C01824=1128.341,-89.185,-46.248,178.702,6.175,149.497
C01825=1128.347,-89.434,-46.238,178.699,6.174,149.498
C01826=1128.352,-89.684,-46.229,178.697,6.174,149.498
C01827=1128.357,-89.934,-46.220,178.696,6.174,149.499
C01828=1128.363,-90.184,-46.210,178.693,6.173,149.499
C01829=1128.368,-90.434,-46.201,178.691,6.172,149.500
C01830=1128.373,-90.683,-46.192,178.690,6.172,149.500
C01831=1128.379,-90.933,-46.182,178.687,6.172,149.501
C01832=1128.384,-91.183,-46.173,178.685,6.171,149.501
C01833=1128.389,-91.433,-46.164,178.683,6.170,149.502
C01834=1128.395,-91.682,-46.154,178.681,6.170,149.502
C01835=1128.400,-91.932,-46.145,178.679,6.169,149.503
C01836=1128.405,-92.182,-46.136,178.677,6.169,149.503
C01837=1128.411,-92.432,-46.127,178.676,6.169,149.504
C01838=1128.416,-92.681,-46.117,178.673,6.168,149.504
C01839=1128.421,-92.930,-46.108,178.671,6.167,149.505
C01840=1128.427,-93.181,-46.099,178.670,6.167,149.505
C01841=1128.433,-93.430,-46.090,178.667,6.166,149.506
C01842=1128.438,-93.680,-46.081,178.665,6.166,149.506
C01843=1128.443,-93.930,-46.071,178.663,6.166,149.507
C01844=1128.448,-94.180,-46.062,178.661,6.165,149.507
C01845=1128.454,-94.430,-46.053,178.659,6.165,149.508
C01846=1128.460,-94.680,-46.044,178.656,6.164,149.508
C01847=1128.465,-94.930,-46.035,178.655,6.164,149.509
C01848=1128.470,-95.179,-46.025,178.653,6.163,149.509
C01849=1128.475,-95.429,-46.016,178.650,6.162,149.510
C01850=1128.481,-95.679,-46.007,178.649,6.162,149.510
C01851=1128.486,-95.929,-45.998,178.647,6.162,149.511
C01852=1128.491,-96.179,-45.989,178.644,6.161,149.511
C01853=1128.497,-96.428,-45.980,178.643,6.161,149.512
C01854=1128.502,-96.677,-45.970,178.641,6.160,149.512
C01855=1128.507,-96.927,-45.961,178.638,6.159,149.513
C01856=1128.513,-97.177,-45.952,178.637,6.160,149.513
C01857=1128.518,-97.427,-45.944,178.635,6.159,149.514
C01858=1128.524,-97.677,-45.934,178.632,6.158,149.514
C01859=1128.529,-97.927,-45.925,178.631,6.158,149.514
C01860=1128.534,-98.177,-45.916,178.629,6.157,149.515
C01861=1128.539,-98.427,-45.907,178.627,6.157,149.515
C01862=1128.546,-98.676,-45.898,178.625,6.157,149.516
C01863=1128.551,-98.926,-45.889,178.623,6.156,149.516
C01864=1128.556,-99.175,-45.880,178.621,6.155,149.517
C01865=1128.561,-99.425,-45.871,178.619,6.155,149.517
C01866=1128.566,-99.675,-45.862,178.617,6.154,149.518
C01867=1128.572,-99.925,-45.852,178.615,6.154,149.518
C01868=1128.577,-100.175,-45.844,178.613,6.154,149.519
C01869=1128.583,-100.424,-45.835,178.611,6.153,149.519
C01870=1128.588,-100.674,-45.826,178.609,6.152,149.520
C01871=1128.593,-100.924,-45.817,178.607,6.152,149.520
C01872=1128.598,-101.173,-45.808,178.605,6.152,149.521
C01873=1128.604,-101.424,-45.799,178.603,6.151,149.521
C01874=1128.609,-101.673,-45.790,178.601,6.151,149.522
C01875=1128.615,-101.923,-45.781,178.599,6.150,149.522
C01876=1128.620,-102.172,-45.772,178.597,6.150,149.523
C01877=1128.626,-102.422,-45.764,178.595,6.149,149.523
C01878=1128.631,-102.672,-45.755,178.593,6.149,149.524
C01879=1128.637,-102.945,-45.745,178.591,6.148,149.524
C01880=1128.642,-103.217,-45.736,178.589,6.148,149.525
C01881=1128.648,-103.489,-45.725,178.586,6.148,149.525
C01882=1128.654,-103.762,-45.715,178.584,6.147,149.526
C01883=1128.660,-104.011,-45.707,178.582,6.146,149.526
C01884=1128.665,-104.261,-45.698,178.580,6.146,149.527
C01885=1128.670,-104.511,-45.689,178.578,6.145,149.527
C01886=1128.676,-104.761,-45.680,178.577,6.145,149.528
C01887=1128.681,-105.011,-45.671,178.574,6.145,149.528
C01888=1128.687,-105.260,-45.663,178.572,6.144,149.529
C01889=1128.692,-105.510,-45.654,178.571,6.144,149.529
C01890=1128.697,-105.760,-45.646,178.568,6.143,149.530
C01891=1128.702,-106.010,-45.637,178.566,6.143,149.530
C01892=1128.708,-106.260,-45.628,178.565,6.143,149.531
C01893=1128.713,-106.509,-45.619,178.562,6.142,149.531
C01894=1128.718,-106.759,-45.610,178.561,6.142,149.532
C01895=1128.724,-107.009,-45.601,178.559,6.141,149.532
C01896=1128.730,-107.259,-45.592,178.556,6.140,149.533
C01897=1128.736,-107.509,-45.584,178.555,6.140,149.533
C01898=1128.741,-107.758,-45.575,178.553,6.140,149.534
C01899=1128.746,-108.008,-45.566,178.551,6.140,149.534
C01900=1128.751,-108.258,-45.557,178.549,6.139,149.535
C01901=1128.757,-108.507,-45.549,178.547,6.138,149.535
C01902=1128.762,-108.757,-45.540,178.545,6.138,149.535
C01903=1128.768,-109.008,-45.532,178.543,6.137,149.536
C01904=1128.773,-109.257,-45.523,178.541,6.136,149.536
C01905=1128.778,-109.507,-45.514,178.539,6.136,149.537
C01906=1128.784,-109.756,-45.506,178.537,6.136,149.537
C01907=1128.789,-110.006,-45.497,178.536,6.136,149.538
C01908=1128.794,-110.257,-45.488,178.533,6.135,149.538
C01909=1128.800,-110.506,-45.480,178.531,6.134,149.539
C01910=1128.805,-110.756,-45.471,178.530,6.134,149.539
C01911=1128.810,-111.006,-45.462,178.527,6.134,149.540
C01912=1128.816,-111.255,-45.454,178.526,6.134,149.540
C01913=1128.822,-111.505,-45.445,178.524,6.133,149.541
C01914=1128.827,-111.755,-45.436,178.521,6.132,149.541
C01915=1128.832,-112.005,-45.428,178.520,6.132,149.542
C01916=1128.838,-112.255,-45.420,178.518,6.131,149.542
C01917=1128.842,-112.504,-45.411,178.516,6.132,149.543
C01918=1128.848,-112.754,-45.403,178.514,6.131,149.543
C01919=1128.853,-113.003,-45.394,178.512,6.131,149.544
C01920=1128.859,-113.254,-45.386,178.510,6.130,149.544
C01921=1128.864,-113.504,-45.377,178.508,6.129,149.545
C01922=1128.870,-113.753,-45.368,178.506,6.129,149.545
C01923=1128.875,-114.003,-45.360,178.505,6.128,149.545
C01924=1128.880,-114.253,-45.351,178.503,6.128,149.546
C01925=1128.886,-114.502,-45.343,178.501,6.128,149.546
C01926=1128.892,-114.753,-45.335,178.499,6.127,149.547
C01927=1128.897,-115.003,-45.326,178.497,6.127,149.547
C01928=1128.903,-115.252,-45.317,178.495,6.126,149.548
C01929=1128.908,-115.502,-45.309,178.493,6.126,149.548
C01930=1128.913,-115.752,-45.300,178.491,6.125,149.549
C01931=1128.918,-116.001,-45.292,178.489,6.125,149.549
C01932=1128.924,-116.251,-45.284,178.487,6.125,149.550
C01933=1128.929,-116.501,-45.275,178.485,6.124,149.550
C01934=1128.935,-116.750,-45.267,178.483,6.124,149.551
C01935=1128.940,-117.001,-45.258,178.481,6.123,149.551
C01936=1128.945,-117.251,-45.249,178.480,6.123,149.552
C01937=1128.951,-117.500,-45.242,178.478,6.122,149.552
C01938=1128.957,-117.750,-45.233,178.476,6.122,149.552
C01939=1128.961,-118.000,-45.224,178.474,6.122,149.553
C01940=1128.967,-118.250,-45.217,178.472,6.121,149.553
C01941=1128.972,-118.499,-45.208,178.470,6.121,149.554
C01942=1128.978,-118.749,-45.200,178.468,6.120,149.554
C01943=1128.983,-118.999,-45.191,178.467,6.120,149.555
C01944=1128.989,-119.250,-45.183,178.464,6.119,149.555
C01945=1128.994,-119.498,-45.175,178.463,6.119,149.556
C01946=1128.999,-119.748,-45.166,178.461,6.119,149.556
C01947=1129.005,-119.999,-45.158,178.459,6.119,149.557
C01948=1129.010,-120.248,-45.149,178.457,6.118,149.557
C01949=1129.016,-120.498,-45.141,178.455,6.117,149.558
C01950=1129.021,-120.747,-45.133,178.453,6.117,149.558
C01951=1129.026,-120.998,-45.125,178.451,6.116,149.559
C01952=1129.032,-121.247,-45.116,178.450,6.116,149.559
C01953=1129.038,-121.497,-45.108,178.447,6.116,149.560
C01954=1129.043,-121.747,-45.099,178.446,6.116,149.560
C01955=1129.048,-121.997,-45.092,178.444,6.115,149.561
C01956=1129.053,-122.246,-45.083,178.442,6.115,149.561
C01957=1129.059,-122.496,-45.075,178.440,6.114,149.562
C01958=1129.064,-122.746,-45.067,178.439,6.114,149.562
C01959=1129.069,-122.996,-45.059,178.436,6.113,149.562
C01960=1129.075,-123.245,-45.050,178.434,6.112,149.563
C01961=1129.080,-123.496,-45.042,178.433,6.112,149.563
C01962=1129.086,-123.745,-45.034,178.430,6.112,149.564
C01963=1129.091,-123.995,-45.026,178.429,6.112,149.564
C01964=1129.097,-124.245,-45.018,178.427,6.111,149.565
C01965=1129.102,-124.495,-45.009,178.425,6.111,149.565
C01966=1129.108,-124.745,-45.001,178.423,6.110,149.565
C01967=1129.113,-124.994,-44.993,178.422,6.110,149.566
C01968=1129.118,-125.244,-44.985,178.420,6.109,149.566
C01969=1129.124,-125.494,-44.977,178.418,6.109,149.567
C01970=1129.129,-125.744,-44.969,178.416,6.109,149.567
C01971=1129.135,-125.994,-44.961,178.414,6.109,149.568
C01972=1129.140,-126.243,-44.952,178.412,6.108,149.568
C01973=1129.146,-126.493,-44.944,178.410,6.108,149.569
C01974=1129.151,-126.743,-44.937,178.409,6.107,149.569
C01975=1129.156,-126.992,-44.928,178.407,6.107,149.570
C01976=1129.162,-127.243,-44.920,178.405,6.106,149.570
C01977=1129.167,-127.492,-44.912,178.403,6.106,149.571
C01978=1129.172,-127.742,-44.904,178.401,6.105,149.571
C01979=1129.179,-127.992,-44.896,178.400,6.105,149.572
C01980=1129.183,-128.242,-44.888,178.397,6.105,149.572
C01981=1129.189,-128.491,-44.880,178.396,6.104,149.572
C01982=1129.195,-128.742,-44.872,178.394,6.104,149.573
C01983=1128.773,-128.753,-44.916,178.391,6.108,149.575
C01984=1128.768,-128.503,-44.925,178.392,6.108,149.574
C01985=1128.762,-128.253,-44.933,178.395,6.108,149.574
C01986=1128.757,-128.003,-44.940,178.396,6.108,149.573
C01987=1128.752,-127.754,-44.949,178.398,6.109,149.573
C01988=1128.746,-127.504,-44.957,178.399,6.109,149.572
C01989=1128.741,-127.254,-44.964,178.402,6.110,149.572
C01990=1128.736,-127.004,-44.973,178.403,6.110,149.571
C01991=1128.730,-126.754,-44.981,178.405,6.111,149.571
C01992=1128.725,-126.504,-44.989,178.407,6.111,149.570
C01993=1128.719,-126.255,-44.997,178.409,6.111,149.570
C01994=1128.714,-126.005,-45.005,178.411,6.111,149.570
C01995=1128.708,-125.755,-45.013,178.413,6.113,149.569
C01996=1128.703,-125.505,-45.021,178.414,6.113,149.569
C01997=1128.697,-125.256,-45.029,178.416,6.113,149.568
C01998=1128.692,-125.006,-45.038,178.418,6.113,149.568
C01999=1128.687,-124.756,-45.046,178.420,6.114,149.567
C02000=1128.681,-124.506,-45.054,178.422,6.114,149.567
C02001=1128.676,-124.256,-45.062,178.424,6.115,149.566
C02002=1128.670,-124.006,-45.070,178.425,6.115,149.566
C02003=1128.665,-123.757,-45.079,178.427,6.116,149.566
C02004=1128.659,-123.507,-45.086,178.429,6.116,149.565
C02005=1128.654,-123.257,-45.095,178.431,6.116,149.565
C02006=1128.648,-123.007,-45.103,178.433,6.117,149.564
C02007=1128.644,-122.758,-45.111,178.435,6.117,149.564
C02008=1128.638,-122.507,-45.120,178.437,6.118,149.563
C02009=1128.632,-122.258,-45.128,178.439,6.118,149.563
C02010=1128.627,-122.008,-45.136,178.441,6.119,149.562
C02011=1128.622,-121.759,-45.144,178.442,6.119,149.562
C02012=1128.617,-121.508,-45.152,178.444,6.120,149.561
C02013=1128.611,-121.258,-45.161,178.446,6.120,149.561
C02014=1128.605,-121.009,-45.169,178.448,6.120,149.560
C02015=1128.601,-120.759,-45.177,178.450,6.121,149.560
C02016=1128.595,-120.509,-45.185,178.452,6.121,149.559
C02017=1128.590,-120.260,-45.194,178.454,6.122,149.559
C02018=1128.584,-120.009,-45.202,178.456,6.122,149.558
C02019=1128.578,-119.760,-45.211,178.458,6.122,149.558
C02020=1128.573,-119.509,-45.219,178.459,6.123,149.558
C02021=1128.568,-119.261,-45.227,178.461,6.124,149.557
C02022=1128.562,-119.010,-45.235,178.463,6.123,149.557
C02023=1128.557,-118.760,-45.244,178.465,6.124,149.556
C02024=1128.551,-118.511,-45.253,178.467,6.125,149.556
C02025=1128.546,-118.261,-45.261,178.469,6.125,149.555
C02026=1128.542,-118.011,-45.269,178.471,6.126,149.555
C02027=1128.535,-117.761,-45.277,178.472,6.126,149.554
C02028=1128.530,-117.512,-45.286,178.475,6.126,149.554
C02029=1128.524,-117.262,-45.294,178.476,6.126,149.553
C02030=1128.519,-117.012,-45.303,178.478,6.127,149.553
C02031=1128.514,-116.762,-45.311,178.480,6.127,149.553
C02032=1128.508,-116.512,-45.319,178.482,6.128,149.552
C02033=1128.503,-116.262,-45.328,178.484,6.129,149.552
C02034=1128.498,-116.013,-45.336,178.486,6.129,149.551
C02035=1128.492,-115.763,-45.344,178.488,6.130,149.551
C02036=1128.487,-115.513,-45.353,178.489,6.129,149.550
C02037=1128.482,-115.263,-45.361,178.492,6.130,149.550
C02038=1128.476,-115.014,-45.370,178.493,6.130,149.549
C02039=1128.471,-114.764,-45.379,178.495,6.131,149.549
C02040=1128.465,-114.513,-45.387,178.498,6.132,149.548
C02041=1128.459,-114.264,-45.395,178.499,6.132,149.548
C02042=1128.454,-114.014,-45.404,178.501,6.132,149.547
C02043=1128.449,-113.764,-45.413,178.503,6.132,149.547
C02044=1128.443,-113.515,-45.421,178.505,6.133,149.546
C02045=1128.438,-113.265,-45.430,178.507,6.134,149.546
C02046=1128.433,-113.015,-45.438,178.508,6.134,149.546
C02047=1128.427,-112.766,-45.446,178.511,6.135,149.545
C02048=1128.422,-112.516,-45.455,178.512,6.135,149.545
C02049=1128.417,-112.266,-45.464,178.514,6.136,149.544
C02050=1128.411,-112.016,-45.472,178.516,6.136,149.544
C02051=1128.406,-111.766,-45.481,178.518,6.136,149.543
C02052=1128.401,-111.516,-45.490,178.520,6.137,149.543
C02053=1128.395,-111.267,-45.498,178.522,6.137,149.542
C02054=1128.389,-111.017,-45.506,178.524,6.138,149.542
C02055=1128.384,-110.767,-45.515,178.526,6.138,149.541
C02056=1128.379,-110.517,-45.524,178.528,6.138,149.541
C02057=1128.373,-110.268,-45.533,178.530,6.139,149.540
C02058=1128.368,-110.018,-45.541,178.532,6.139,149.540
C02059=1128.363,-109.768,-45.550,178.534,6.140,149.539
C02060=1128.357,-109.518,-45.559,178.536,6.140,149.539
C02061=1128.352,-109.269,-45.567,178.538,6.141,149.538
C02062=1128.346,-109.019,-45.576,178.540,6.141,149.538
C02063=1128.341,-108.769,-45.585,178.542,6.141,149.537
C02064=1128.336,-108.518,-45.593,178.544,6.142,149.537
C02065=1128.330,-108.269,-45.602,178.546,6.143,149.536
C02066=1128.325,-108.019,-45.610,178.547,6.143,149.536
C02067=1128.320,-107.770,-45.619,178.549,6.144,149.536
C02068=1128.315,-107.520,-45.628,178.551,6.144,149.535
C02069=1128.309,-107.271,-45.637,178.553,6.144,149.535
C02070=1128.303,-107.020,-45.645,178.555,6.145,149.534
C02071=1128.298,-106.770,-45.654,178.557,6.145,149.534
C02072=1128.293,-106.520,-45.663,178.559,6.146,149.533
C02073=1128.287,-106.271,-45.671,178.561,6.146,149.533
C02074=1128.282,-106.021,-45.680,178.563,6.147,149.532
C02075=1128.276,-105.771,-45.690,178.565,6.147,149.532
C02076=1128.271,-105.521,-45.699,178.567,6.147,149.531
C02077=1128.266,-105.272,-45.707,178.569,6.148,149.531
C02078=1128.260,-105.022,-45.716,178.571,6.149,149.530
C02079=1128.255,-104.772,-45.724,178.573,6.149,149.530
C02080=1128.249,-104.522,-45.733,178.575,6.149,149.529
C02081=1128.244,-104.272,-45.742,178.576,6.149,149.529
C02082=1128.239,-104.022,-45.751,178.579,6.150,149.528
C02083=1128.233,-103.773,-45.759,178.581,6.151,149.528
C02084=1128.228,-103.501,-45.769,178.583,6.152,149.527
C02085=1128.222,-103.229,-45.779,178.585,6.152,149.527
C02086=1128.216,-102.956,-45.789,178.587,6.152,149.526
C02087=1128.210,-102.684,-45.798,178.590,6.153,149.526
C02088=1128.205,-102.433,-45.808,178.592,6.153,149.525
C02089=1128.199,-102.184,-45.817,178.593,6.153,149.525
C02090=1128.194,-101.934,-45.825,178.596,6.154,149.524
C02091=1128.188,-101.685,-45.834,178.597,6.154,149.524
C02092=1128.183,-101.435,-45.843,178.599,6.155,149.523
C02093=1128.178,-101.185,-45.852,178.602,6.156,149.523
C02094=1128.173,-100.935,-45.861,178.603,6.156,149.522
C02095=1128.167,-100.685,-45.870,178.605,6.156,149.522
C02096=1128.162,-100.435,-45.879,178.608,6.157,149.521
C02097=1128.156,-100.186,-45.888,178.609,6.157,149.521
C02098=1128.151,-99.936,-45.897,178.611,6.158,149.520
C02099=1128.146,-99.686,-45.905,178.614,6.158,149.520
C02100=1128.140,-99.436,-45.915,178.615,6.158,149.519
C02101=1128.135,-99.186,-45.924,178.617,6.159,149.519
C02102=1128.130,-98.937,-45.933,178.620,6.160,149.518
C02103=1128.125,-98.687,-45.942,178.621,6.160,149.518
C02104=1128.119,-98.438,-45.951,178.623,6.161,149.517
C02105=1128.113,-98.188,-45.960,178.626,6.161,149.517
C02106=1128.108,-97.938,-45.969,178.627,6.161,149.516
C02107=1128.103,-97.688,-45.978,178.629,6.162,149.516
C02108=1128.097,-97.438,-45.987,178.631,6.163,149.515
C02109=1128.092,-97.188,-45.996,178.633,6.163,149.515
C02110=1128.086,-96.938,-46.005,178.635,6.164,149.514
C02111=1128.081,-96.688,-46.014,178.637,6.164,149.514
C02112=1128.076,-96.440,-46.024,178.639,6.164,149.513
C02113=1128.071,-96.190,-46.032,178.641,6.165,149.513
C02114=1128.065,-95.940,-46.042,178.643,6.166,149.512
C02115=1128.060,-95.690,-46.051,178.645,6.166,149.512
C02116=1128.054,-95.440,-46.060,178.647,6.166,149.511
C02117=1128.048,-95.190,-46.069,178.649,6.167,149.511
C02118=1128.043,-94.940,-46.078,178.651,6.167,149.510
C02119=1128.038,-94.691,-46.088,178.653,6.168,149.510
C02120=1128.033,-94.441,-46.097,178.655,6.169,149.509
C02121=1128.027,-94.191,-46.106,178.657,6.169,149.509
C02122=1128.022,-93.941,-46.115,178.659,6.169,149.509
C02123=1128.017,-93.691,-46.124,178.661,6.170,149.508
C02124=1128.011,-93.442,-46.134,178.664,6.171,149.508
C02125=1128.006,-93.192,-46.143,178.665,6.171,149.507
C02126=1128.001,-92.943,-46.152,178.667,6.172,149.507
C02127=1127.995,-92.692,-46.161,178.670,6.172,149.506
C02128=1127.990,-92.443,-46.171,178.672,6.172,149.505
C02129=1127.985,-92.193,-46.180,178.674,6.173,149.505
C02130=1127.979,-91.943,-46.189,178.676,6.173,149.504
C02131=1127.974,-91.693,-46.198,178.678,6.173,149.504
C02132=1127.969,-91.444,-46.208,178.680,6.174,149.503
C02133=1127.963,-91.194,-46.217,178.682,6.175,149.503
C02134=1127.958,-90.944,-46.226,178.684,6.176,149.502
C02135=1127.952,-90.694,-46.235,178.686,6.176,149.502
C02136=1127.947,-90.445,-46.245,178.688,6.176,149.502
C02137=1127.942,-90.195,-46.254,178.690,6.177,149.501
C02138=1127.936,-89.945,-46.263,178.692,6.177,149.501
C02139=1127.931,-89.695,-46.273,178.694,6.178,149.500
C02140=1127.926,-89.446,-46.282,178.696,6.178,149.500
C02141=1127.921,-89.196,-46.291,178.698,6.179,149.499
C02142=1127.915,-88.946,-46.301,178.700,6.179,149.499
C02143=1127.910,-88.696,-46.310,178.702,6.180,149.498
C02144=1127.904,-88.446,-46.320,178.704,6.181,149.498
C02145=1127.899,-88.197,-46.329,178.706,6.181,149.497
C02146=1127.894,-87.947,-46.338,178.708,6.181,149.497
C02147=1127.888,-87.697,-46.348,178.711,6.182,149.496
C02148=1127.883,-87.448,-46.357,178.713,6.182,149.495
C02149=1127.877,-87.198,-46.367,178.715,6.182,149.495
C02150=1127.872,-86.948,-46.376,178.717,6.183,149.494
C02151=1127.866,-86.698,-46.386,178.719,6.184,149.494
C02152=1127.861,-86.448,-46.395,178.721,6.184,149.494
C02153=1127.856,-86.199,-46.404,178.723,6.185,149.493
C02154=1127.850,-85.949,-46.414,178.725,6.185,149.493
C02155=1127.846,-85.700,-46.423,178.727,6.186,149.492
C02156=1127.840,-85.449,-46.433,178.729,6.186,149.492
C02157=1127.835,-85.200,-46.443,178.731,6.187,149.491
C02158=1127.830,-84.949,-46.452,178.733,6.188,149.491
C02159=1127.824,-84.700,-46.461,178.735,6.188,149.490
C02160=1127.819,-84.450,-46.471,178.737,6.188,149.490
C02161=1127.814,-84.200,-46.480,178.740,6.189,149.489
C02162=1127.808,-83.951,-46.491,178.742,6.189,149.488
C02163=1127.803,-83.701,-46.499,178.744,6.190,149.488
C02164=1127.797,-83.451,-46.510,178.746,6.190,149.487
C02165=1127.792,-83.201,-46.519,178.748,6.191,149.487
C02166=1127.786,-82.952,-46.529,178.750,6.192,149.487
C02167=1127.781,-82.702,-46.538,178.752,6.192,149.486
C02168=1127.776,-82.452,-46.548,178.754,6.192,149.486
C02169=1127.771,-82.203,-46.557,178.756,6.193,149.485
C02170=1127.766,-81.952,-46.567,178.758,6.194,149.485
C02171=1127.760,-81.702,-46.576,178.760,6.195,149.484
C02172=1127.755,-81.453,-46.586,178.763,6.194,149.483
C02173=1127.750,-81.203,-46.595,178.765,6.195,149.483
C02174=1127.744,-80.954,-46.606,178.767,6.196,149.482
C02175=1127.739,-80.704,-46.615,178.769,6.196,149.482
C02176=1127.733,-80.454,-46.625,178.771,6.196,149.481
C02177=1127.728,-80.205,-46.635,178.773,6.197,149.481
C02178=1127.723,-79.955,-46.644,178.775,6.198,149.480
C02179=1127.718,-79.705,-46.654,178.777,6.199,149.480
C02180=1127.713,-79.455,-46.664,178.779,6.199,149.480
C02181=1127.707,-79.205,-46.673,178.781,6.199,149.479
C02182=1127.702,-78.956,-46.683,178.783,6.200,149.479
C02183=1127.696,-78.706,-46.693,178.786,6.201,149.478
C02184=1127.690,-78.456,-46.703,178.788,6.201,149.477
C02185=1127.686,-78.207,-46.712,178.790,6.201,149.477
C02186=1127.680,-77.957,-46.722,178.792,6.202,149.476
C02187=1127.675,-77.707,-46.732,178.794,6.203,149.476
C02188=1127.669,-77.435,-46.742,178.796,6.204,149.475
C02189=1127.663,-77.164,-46.753,178.799,6.204,149.475
C02190=1127.657,-76.892,-46.764,178.801,6.205,149.474
C02191=1127.652,-76.621,-46.775,178.803,6.205,149.474
C02192=1127.646,-76.370,-46.784,178.805,6.205,149.473
C02193=1127.641,-76.121,-46.794,178.807,6.206,149.473
C02194=1127.636,-75.872,-46.804,178.809,6.207,149.472
C02195=1127.630,-75.621,-46.814,178.812,6.207,149.472
C02196=1127.621,-75.201,-46.831,178.815,6.208,149.471
C02197=1127.594,-73.952,-46.879,179.491,4.912,148.990
C02198=1127.589,-73.702,-46.889,179.491,4.918,148.991
C02199=1127.584,-73.452,-46.898,179.492,4.923,148.992
C02200=1127.578,-73.203,-46.908,179.492,4.928,148.993
C02201=1127.573,-72.953,-46.917,179.492,4.934,148.994
C02202=1127.567,-72.703,-46.927,179.493,4.939,148.995
C02203=1127.563,-72.453,-46.937,179.493,4.945,148.996
C02204=1127.557,-72.203,-46.947,179.493,4.950,148.998
C02205=1127.551,-71.953,-46.956,179.493,4.955,148.999
C02206=1127.546,-71.704,-46.966,179.494,4.961,149.000
C02207=1127.540,-71.454,-46.975,179.494,4.965,149.001
C02208=1127.535,-71.205,-46.985,179.494,4.971,149.002
C02209=1127.530,-70.955,-46.995,179.495,4.976,149.003
C02210=1127.525,-70.705,-47.004,179.495,4.981,149.004
C02211=1127.519,-70.456,-47.014,179.495,4.987,149.005
C02212=1127.514,-70.205,-47.024,179.496,4.992,149.006
C02213=1127.509,-69.956,-47.034,179.497,4.998,149.007
C02214=1127.503,-69.706,-47.044,179.496,5.003,149.008
C02215=1127.497,-69.456,-47.053,179.497,5.008,149.009
C02216=1127.493,-69.207,-47.063,179.497,5.014,149.010
C02217=1127.487,-68.957,-47.073,179.498,5.019,149.011
C02218=1127.481,-68.707,-47.083,179.498,5.024,149.012
C02219=1127.477,-68.457,-47.093,179.499,5.030,149.013
C02220=1127.471,-68.207,-47.103,179.499,5.035,149.014
C02221=1127.466,-67.958,-47.113,179.500,5.041,149.015
C02222=1127.460,-67.708,-47.122,179.500,5.045,149.016
C02223=1127.455,-67.458,-47.132,179.501,5.051,149.017
C02224=1127.450,-67.208,-47.143,179.502,5.057,149.018
C02225=1127.445,-66.959,-47.152,179.502,5.062,149.019
C02226=1127.439,-66.709,-47.162,179.503,5.067,149.020
C02227=1127.433,-66.459,-47.172,179.503,5.072,149.021
C02228=1127.428,-66.210,-47.182,179.504,5.078,149.022
C02229=1127.424,-65.960,-47.192,179.505,5.084,149.023
C02230=1127.418,-65.710,-47.203,179.505,5.088,149.024
C02231=1127.412,-65.460,-47.212,179.506,5.094,149.025
C02232=1127.407,-65.211,-47.222,179.507,5.099,149.026
C02233=1127.402,-64.961,-47.232,179.507,5.105,149.027
C02234=1127.397,-64.711,-47.242,179.508,5.110,149.028
C02235=1127.391,-64.462,-47.253,179.509,5.116,149.029
C02236=1127.385,-64.212,-47.263,179.509,5.120,149.030
C02237=1127.381,-63.962,-47.273,179.510,5.126,149.030
C02238=1127.375,-63.712,-47.282,179.511,5.132,149.031
C02239=1127.370,-63.462,-47.293,179.512,5.136,149.032
C02240=1127.365,-63.212,-47.303,179.513,5.142,149.033
C02241=1127.359,-62.963,-47.313,179.514,5.148,149.034
C02242=1127.354,-62.713,-47.324,179.515,5.153,149.035
C02243=1127.349,-62.464,-47.333,179.515,5.158,149.036
C02244=1127.344,-62.214,-47.344,179.516,5.163,149.037
C02245=1127.338,-61.964,-47.354,179.517,5.169,149.038
C02246=1127.329,-61.547,-47.372,179.519,5.178,149.039
C02247=1127.321,-61.128,-47.388,179.520,5.187,149.041
C02248=1127.311,-60.711,-47.405,179.522,5.196,149.042
C02249=1127.303,-60.293,-47.423,179.524,5.204,149.043
C02250=1127.297,-60.043,-47.433,179.524,5.210,149.045
C02251=1127.292,-59.794,-47.444,179.523,5.214,149.046
C02252=1127.287,-59.543,-47.454,179.523,5.219,149.047
C02253=1127.281,-59.294,-47.464,179.523,5.223,149.048
C02254=1127.275,-59.044,-47.475,179.523,5.228,149.049
C02255=1127.271,-58.795,-47.486,179.522,5.232,149.050
C02256=1127.265,-58.545,-47.496,179.522,5.237,149.051
C02257=1127.261,-58.295,-47.506,179.522,5.241,149.052
C02258=1127.255,-58.046,-47.516,179.522,5.246,149.053
C02259=1127.250,-57.796,-47.527,179.521,5.251,149.054
C02260=1127.245,-57.546,-47.537,179.522,5.255,149.055
C02261=1127.239,-57.296,-47.547,179.521,5.261,149.056
C02262=1127.234,-57.047,-47.559,179.521,5.265,149.057
C02263=1127.229,-56.797,-47.569,179.521,5.270,149.058
C02264=1127.224,-56.547,-47.579,179.520,5.274,149.059
C02265=1127.218,-56.297,-47.590,179.520,5.279,149.061
C02266=1127.213,-56.048,-47.600,179.520,5.283,149.062
C02267=1127.208,-55.797,-47.610,179.520,5.288,149.063
C02268=1127.202,-55.549,-47.621,179.519,5.293,149.064
C02269=1127.197,-55.298,-47.632,179.520,5.297,149.065
C02270=1127.192,-55.049,-47.642,179.519,5.302,149.066
C02271=1127.187,-54.798,-47.653,179.519,5.307,149.067
C02272=1127.181,-54.550,-47.664,179.519,5.312,149.068
C02273=1127.176,-54.300,-47.674,179.519,5.316,149.069
C02274=1127.170,-54.049,-47.685,179.519,5.321,149.070
C02275=1127.165,-53.800,-47.695,179.518,5.325,149.071
C02276=1127.160,-53.550,-47.706,179.518,5.330,149.072
C02277=1127.154,-53.301,-47.717,179.518,5.335,149.073
C02278=1127.149,-53.051,-47.727,179.518,5.339,149.074
C02279=1127.144,-52.801,-47.737,179.517,5.344,149.076
C02280=1127.139,-52.551,-47.749,179.517,5.349,149.077
C02281=1127.133,-52.302,-47.759,179.517,5.354,149.078
C02282=1127.128,-52.052,-47.770,179.517,5.358,149.079
C02283=1127.123,-51.803,-47.780,179.517,5.363,149.080
C02284=1127.118,-51.552,-47.791,179.516,5.367,149.081
C02285=1127.112,-51.303,-47.801,179.517,5.372,149.082
C02286=1127.107,-51.053,-47.813,179.516,5.377,149.083
C02287=1127.101,-50.803,-47.823,179.516,5.382,149.084
C02288=1127.096,-50.553,-47.834,179.516,5.386,149.085
C02289=1127.091,-50.304,-47.845,179.516,5.391,149.086
C02290=1127.086,-50.054,-47.855,179.516,5.396,149.087
C02291=1127.081,-49.805,-47.866,179.515,5.400,149.089
C02292=1127.076,-49.555,-47.877,179.515,5.405,149.089
C02293=1127.070,-49.305,-47.888,179.515,5.409,149.091
C02294=1127.065,-49.055,-47.899,179.515,5.415,149.092
C02295=1127.059,-48.806,-47.909,179.514,5.418,149.093
C02296=1127.055,-48.556,-47.921,179.514,5.424,149.094
C02297=1127.049,-48.307,-47.931,179.514,5.429,149.095
C02298=1127.044,-48.091,-47.940,179.514,5.433,149.096
C02299=1127.040,-47.875,-47.950,179.514,5.437,149.097
C02300=1127.036,-47.659,-47.959,179.514,5.441,149.098
C02301=1127.031,-47.444,-47.968,179.514,5.445,149.099
C02302=1127.026,-47.228,-47.978,179.513,5.449,149.100
C02303=1127.022,-47.013,-47.987,179.513,5.453,149.100
C02304=1127.017,-46.797,-47.996,179.513,5.456,149.101
C02305=1127.012,-46.582,-48.005,179.513,5.460,149.102
C02306=1127.007,-46.332,-48.017,179.513,5.466,149.103
C02307=1127.002,-46.082,-48.028,179.512,5.470,149.105
C02308=1126.997,-45.833,-48.039,179.512,5.475,149.106
C02309=1126.992,-45.583,-48.049,179.513,5.480,149.107
C02310=1126.986,-45.333,-48.061,179.512,5.484,149.108
C02311=1126.981,-45.083,-48.071,179.512,5.489,149.109
C02312=1126.975,-44.834,-48.082,179.511,5.494,149.110
C02313=1126.970,-44.584,-48.093,179.512,5.498,149.111
C02314=1126.965,-44.334,-48.105,179.511,5.504,149.112
C02315=1126.959,-44.084,-48.115,179.511,5.508,149.113
C02316=1126.955,-43.835,-48.126,179.511,5.513,149.114
C02317=1126.949,-43.585,-48.137,179.511,5.517,149.115
C02318=1126.944,-43.335,-48.148,179.511,5.522,149.116
C02319=1126.939,-43.086,-48.160,179.511,5.527,149.117
C02320=1126.933,-42.836,-48.170,179.513,5.533,149.118
C02321=1126.928,-42.586,-48.182,179.515,5.539,149.119
C02322=1126.922,-42.337,-48.192,179.517,5.545,149.120
C02323=1126.918,-42.087,-48.203,179.518,5.550,149.120
C02324=1126.912,-41.837,-48.215,179.521,5.556,149.121
C02325=1126.907,-41.588,-48.225,179.523,5.562,149.121
C02326=1126.902,-41.338,-48.237,179.524,5.567,149.122
C02327=1126.896,-41.088,-48.249,179.526,5.573,149.123
C02328=1126.891,-40.838,-48.259,179.527,5.579,149.124
C02329=1126.886,-40.589,-48.270,179.529,5.585,149.124
C02330=1126.881,-40.339,-48.282,179.531,5.590,149.125
C02331=1126.875,-40.090,-48.293,179.533,5.595,149.126
C02332=1126.870,-39.839,-48.304,179.534,5.601,149.127
C02333=1126.865,-39.590,-48.315,179.535,5.606,149.127
C02334=1126.860,-39.340,-48.327,179.537,5.611,149.128
C02335=1126.854,-39.091,-48.338,179.538,5.616,149.129
C02336=1126.849,-38.841,-48.350,179.539,5.622,149.129
C02337=1126.844,-38.591,-48.361,179.541,5.627,149.130
C02338=1126.838,-38.342,-48.372,179.542,5.632,149.131
C02339=1126.833,-38.092,-48.383,179.543,5.638,149.132
C02340=1126.828,-37.842,-48.395,179.545,5.643,149.132
C02341=1126.823,-37.592,-48.407,179.546,5.647,149.133
C02342=1126.817,-37.343,-48.418,179.547,5.653,149.134
C02343=1126.812,-37.094,-48.429,179.548,5.657,149.135
C02344=1126.807,-36.844,-48.441,179.549,5.663,149.135
C02345=1126.802,-36.594,-48.453,179.550,5.667,149.136
C02346=1126.796,-36.343,-48.464,179.551,5.672,149.137
C02347=1126.791,-36.094,-48.475,179.552,5.677,149.138
C02348=1126.786,-35.845,-48.487,179.552,5.682,149.139
C02349=1126.781,-35.595,-48.498,179.553,5.686,149.139
C02350=1126.776,-35.345,-48.510,179.554,5.691,149.140
C02351=1126.770,-35.095,-48.522,179.555,5.696,149.141
C02352=1126.765,-34.846,-48.533,179.556,5.701,149.142
C02353=1126.759,-34.596,-48.544,179.556,5.705,149.143
C02354=1126.756,-34.381,-48.555,179.556,5.709,149.143
C02355=1126.751,-34.165,-48.564,179.557,5.712,149.144
C02356=1126.746,-33.950,-48.575,179.558,5.717,149.145
C02357=1126.742,-33.734,-48.585,179.558,5.721,149.146
C02358=1126.738,-33.519,-48.594,179.558,5.724,149.146
C02359=1126.733,-33.304,-48.605,179.558,5.728,149.147
C02360=1126.728,-33.087,-48.615,179.559,5.733,149.148
C02361=1126.723,-32.872,-48.625,179.559,5.736,149.148
C02362=1126.719,-32.623,-48.637,179.559,5.740,149.149
C02363=1126.713,-32.373,-48.648,179.559,5.745,149.150
C02364=1126.709,-32.123,-48.660,179.559,5.749,149.151
C02365=1126.703,-31.873,-48.672,179.560,5.754,149.152
C02366=1126.697,-31.624,-48.683,179.560,5.758,149.153
C02367=1126.693,-31.375,-48.695,179.559,5.761,149.154
C02368=1126.687,-31.125,-48.707,179.559,5.767,149.155
C02369=1126.682,-30.875,-48.719,179.559,5.771,149.156
C02370=1126.676,-30.625,-48.731,179.559,5.774,149.157
C02371=1126.672,-30.375,-48.742,179.559,5.778,149.158
C02372=1126.666,-30.126,-48.754,179.558,5.783,149.159
C02373=1126.661,-29.876,-48.766,179.558,5.787,149.160
C02374=1126.656,-29.627,-48.778,179.558,5.791,149.161
C02375=1126.650,-29.377,-48.789,179.557,5.795,149.162
C02376=1126.645,-29.127,-48.801,179.557,5.799,149.163
C02377=1126.640,-28.878,-48.813,179.557,5.803,149.164
C02378=1126.635,-28.628,-48.824,179.556,5.808,149.165
C02379=1126.630,-28.379,-48.837,179.555,5.811,149.166
C02380=1126.624,-28.129,-48.849,179.555,5.815,149.167
C02381=1126.620,-27.879,-48.860,179.554,5.819,149.168
C02382=1126.614,-27.629,-48.872,179.553,5.823,149.169
C02383=1126.609,-27.379,-48.884,179.552,5.827,149.170
C02384=1126.604,-27.130,-48.896,179.551,5.831,149.172
C02385=1126.599,-26.880,-48.908,179.550,5.835,149.173
C02386=1126.593,-26.631,-48.919,179.549,5.839,149.174
C02387=1126.588,-26.381,-48.931,179.548,5.843,149.175
C02388=1126.583,-26.131,-48.943,179.547,5.847,149.176
C02389=1126.578,-25.882,-48.955,179.547,5.851,149.177
C02390=1126.572,-25.632,-48.967,179.548,5.856,149.178
C02391=1126.567,-25.382,-48.979,179.548,5.861,149.179
C02392=1126.562,-25.133,-48.990,179.549,5.866,149.180
C02393=1126.557,-24.883,-49.003,179.550,5.871,149.181
C02394=1126.552,-24.633,-49.015,179.551,5.876,149.181
C02395=1126.546,-24.383,-49.027,179.552,5.881,149.182
C02396=1126.541,-24.134,-49.039,179.552,5.886,149.183
C02397=1126.536,-23.884,-49.050,179.553,5.891,149.184
C02398=1126.531,-23.634,-49.062,179.554,5.896,149.185
C02399=1126.526,-23.385,-49.075,179.555,5.901,149.186
C02400=1126.520,-23.135,-49.087,179.555,5.905,149.187
C02401=1126.515,-22.885,-49.099,179.556,5.911,149.187
C02402=1126.510,-22.636,-49.111,179.557,5.915,149.188
C02403=1126.504,-22.386,-49.123,179.558,5.920,149.189
C02404=1126.500,-22.136,-49.134,179.558,5.925,149.190
C02405=1126.495,-21.887,-49.147,179.559,5.930,149.191
C02406=1126.489,-21.637,-49.159,179.560,5.935,149.192
C02407=1126.484,-21.388,-49.172,179.561,5.939,149.192
C02408=1126.479,-21.138,-49.183,179.562,5.945,149.193
C02409=1126.473,-20.889,-49.196,179.562,5.950,149.194
C02410=1126.469,-20.674,-49.206,179.563,5.953,149.195
C02411=1126.465,-20.458,-49.217,179.564,5.958,149.195
C02412=1126.460,-20.243,-49.228,179.565,5.962,149.196
C02413=1126.456,-20.026,-49.237,179.565,5.966,149.197
C02414=1126.450,-19.811,-49.248,179.566,5.970,149.198
C02415=1126.447,-19.596,-49.258,179.567,5.975,149.198
C02416=1126.442,-19.381,-49.269,179.567,5.978,149.199
C02417=1126.437,-19.165,-49.280,179.567,5.983,149.200
C02418=1126.432,-18.915,-49.292,179.568,5.987,149.201
C02419=1126.427,-18.666,-49.305,179.569,5.992,149.201
C02420=1126.421,-18.416,-49.317,179.570,5.998,149.202
C02421=1126.416,-18.167,-49.330,179.571,6.002,149.203
C02422=1126.411,-17.917,-49.341,179.571,6.007,149.204
C02423=1126.406,-17.667,-49.354,179.572,6.011,149.205
C02424=1126.400,-17.418,-49.366,179.573,6.016,149.205
C02425=1126.395,-17.168,-49.378,179.573,6.020,149.206
C02426=1126.391,-16.918,-49.391,179.574,6.026,149.207
C02427=1126.385,-16.668,-49.403,179.575,6.030,149.208
C02428=1126.380,-16.419,-49.416,179.576,6.035,149.209
C02429=1126.375,-16.170,-49.429,179.576,6.040,149.210
C02430=1126.370,-15.920,-49.440,179.577,6.044,149.211
C02431=1126.365,-15.670,-49.453,179.578,6.049,149.211
C02432=1126.359,-15.420,-49.465,179.578,6.054,149.212
C02433=1126.354,-15.171,-49.478,179.579,6.059,149.213
C02434=1126.349,-14.921,-49.490,179.580,6.063,149.214
C02435=1126.344,-14.672,-49.503,179.581,6.068,149.215
C02436=1126.339,-14.422,-49.515,179.581,6.073,149.215
C02437=1126.334,-14.173,-49.528,179.582,6.077,149.216
C02438=1126.329,-13.923,-49.540,179.583,6.082,149.217
C02439=1126.323,-13.673,-49.552,179.583,6.087,149.218
C02440=1126.318,-13.423,-49.566,179.584,6.091,149.219
C02441=1126.313,-13.174,-49.578,179.585,6.096,149.219
C02442=1126.308,-12.924,-49.591,179.585,6.101,149.220
C02443=1126.303,-12.675,-49.603,179.586,6.105,149.221
C02444=1126.297,-12.425,-49.615,179.587,6.110,149.222
C02445=1126.293,-12.175,-49.628,179.588,6.115,149.223
C02446=1126.287,-11.926,-49.641,179.589,6.119,149.223
C02447=1126.282,-11.676,-49.654,179.589,6.124,149.224
C02448=1126.277,-11.427,-49.667,179.590,6.129,149.225
C02449=1126.271,-11.177,-49.679,179.591,6.133,149.226
C02450=1126.267,-10.927,-49.692,179.591,6.138,149.227
C02451=1126.261,-10.678,-49.704,179.592,6.142,149.227
C02452=1126.256,-10.428,-49.717,179.593,6.147,149.228
C02453=1126.250,-10.179,-49.730,179.593,6.152,149.229
C02454=1126.246,-9.929,-49.743,179.594,6.156,149.230
C02455=1126.241,-9.679,-49.755,179.595,6.161,149.231
C02456=1126.236,-9.430,-49.768,179.595,6.166,149.232
C02457=1126.230,-9.180,-49.781,179.596,6.170,149.232
C02458=1126.225,-8.930,-49.794,179.597,6.175,149.233
C02459=1126.220,-8.680,-49.806,179.597,6.179,149.234
C02460=1126.215,-8.431,-49.819,179.598,6.184,149.235
C02461=1126.210,-8.181,-49.832,179.599,6.188,149.236
C02462=1126.204,-7.931,-49.845,179.599,6.193,149.236
C02463=1126.199,-7.682,-49.857,179.600,6.198,149.237
C02464=1126.194,-7.433,-49.870,179.600,6.201,149.238
C02465=1126.189,-7.182,-49.884,179.601,6.206,149.239
C02466=1126.185,-6.968,-49.894,179.602,6.211,149.240
C02467=1126.180,-6.752,-49.905,179.602,6.214,149.240
C02468=1126.176,-6.537,-49.917,179.603,6.218,149.241
C02469=1126.171,-6.322,-49.928,179.604,6.222,149.242
C02470=1126.167,-6.107,-49.939,179.604,6.226,149.242
C02471=1126.162,-5.891,-49.950,179.605,6.230,149.243
C02472=1126.158,-5.676,-49.962,179.605,6.234,149.244
C02473=1126.153,-5.460,-49.973,179.606,6.238,149.244
C02474=1126.148,-5.211,-49.985,179.606,6.242,149.245
C02475=1126.143,-4.961,-49.999,179.607,6.246,149.246
C02476=1126.138,-4.711,-50.011,179.607,6.251,149.247
C02477=1126.133,-4.463,-50.025,179.608,6.256,149.248
C02478=1126.128,-4.212,-50.038,179.609,6.260,149.248
C02479=1126.122,-3.963,-50.051,179.609,6.265,149.249
C02480=1126.117,-3.714,-50.063,179.610,6.270,149.250
C02481=1126.112,-3.463,-50.077,179.611,6.274,149.251
C02482=1126.107,-3.214,-50.090,179.611,6.279,149.252
C02483=1126.102,-2.964,-50.103,179.612,6.283,149.253
C02484=1126.097,-2.715,-50.116,179.612,6.287,149.253
C02485=1126.092,-2.466,-50.129,179.613,6.292,149.254
C02486=1126.087,-2.215,-50.143,179.613,6.296,149.255
C02487=1126.081,-1.966,-50.155,179.614,6.301,149.256
C02488=1126.076,-1.716,-50.168,179.615,6.305,149.257
C02489=1126.071,-1.466,-50.181,179.615,6.310,149.257
C02490=1126.065,-1.217,-50.195,179.616,6.315,149.258
C02491=1126.061,-0.967,-50.208,179.616,6.319,149.259
C02492=1126.055,-0.718,-50.221,179.617,6.323,149.260
C02493=1126.051,-0.468,-50.234,179.617,6.328,149.261
C02494=1126.046,-0.219,-50.248,179.618,6.333,149.262
C02495=1126.040,0.031,-50.261,179.618,6.337,149.262
C02496=1126.035,0.281,-50.274,179.619,6.342,149.263
C02497=1126.030,0.530,-50.288,179.620,6.346,149.264
C02498=1126.025,0.780,-50.301,179.620,6.350,149.265
C02499=1126.019,1.029,-50.314,179.620,6.355,149.266
C02500=1126.015,1.279,-50.327,179.621,6.359,149.266
C02501=1126.009,1.528,-50.341,179.622,6.364,149.267
C02502=1126.004,1.778,-50.353,179.623,6.369,149.268
C02503=1125.999,2.028,-50.367,179.622,6.373,149.269
C02504=1125.993,2.277,-50.381,179.623,6.378,149.270
C02505=1125.989,2.527,-50.394,179.624,6.382,149.271
C02506=1125.983,2.776,-50.408,179.625,6.387,149.272
C02507=1125.979,3.026,-50.421,179.625,6.391,149.272
C02508=1125.973,3.276,-50.434,179.625,6.395,149.273
C02509=1125.969,3.525,-50.448,179.626,6.400,149.274
C02510=1125.963,3.775,-50.461,179.626,6.405,149.275
C02511=1125.959,4.024,-50.475,179.627,6.409,149.276
C02512=1125.953,4.274,-50.488,179.628,6.414,149.277
C02513=1125.947,4.524,-50.501,179.628,6.418,149.277
C02514=1125.943,4.773,-50.515,179.628,6.422,149.278
C02515=1125.937,5.023,-50.528,179.629,6.427,149.279
C02516=1125.933,5.272,-50.541,179.629,6.432,149.280
C02517=1125.927,5.522,-50.555,179.630,6.437,149.281
C02518=1125.922,5.771,-50.569,179.630,6.440,149.282
C02519=1125.917,6.021,-50.582,179.631,6.445,149.283
C02520=1125.912,6.270,-50.596,179.631,6.450,149.283
C02521=1125.906,6.521,-50.609,179.632,6.454,149.284
C02522=1125.902,6.736,-50.621,179.632,6.458,149.285
C02523=1125.898,6.951,-50.633,179.632,6.462,149.286
C02524=1125.893,7.166,-50.644,179.632,6.465,149.286
C02525=1125.889,7.381,-50.656,179.633,6.470,149.287
C02526=1125.884,7.596,-50.668,179.633,6.473,149.288
C02527=1125.880,7.812,-50.680,179.634,6.477,149.289
C02528=1125.876,8.027,-50.691,179.634,6.481,149.290
C02529=1125.872,8.242,-50.703,179.635,6.485,149.290
C02530=1125.866,8.492,-50.716,179.635,6.490,149.291
C02531=1125.861,8.742,-50.731,179.636,6.495,149.292
C02532=1125.856,8.990,-50.744,179.637,6.499,149.293
C02533=1125.851,9.241,-50.757,179.637,6.504,149.294
C02534=1125.846,9.490,-50.772,179.639,6.509,149.294
C02535=1125.841,9.739,-50.785,179.640,6.514,149.295
C02536=1125.836,9.989,-50.799,179.640,6.518,149.296
C02537=1125.830,10.238,-50.812,179.641,6.523,149.297
C02538=1125.825,10.489,-50.826,179.642,6.527,149.297
C02539=1125.821,10.738,-50.840,179.642,6.532,149.298
C02540=1125.815,10.987,-50.854,179.644,6.537,149.299
C02541=1125.810,11.237,-50.867,179.645,6.542,149.300
C02542=1125.804,11.486,-50.881,179.646,6.546,149.301
C02543=1125.799,11.736,-50.895,179.646,6.551,149.301
C02544=1125.795,11.986,-50.909,179.647,6.555,149.302
C02545=1125.789,12.235,-50.922,179.648,6.560,149.303
C02546=1125.784,12.485,-50.937,179.649,6.565,149.304
C02547=1125.779,12.735,-50.951,179.650,6.570,149.304
C02548=1125.774,12.984,-50.965,179.651,6.574,149.305
C02549=1125.769,13.234,-50.978,179.651,6.579,149.306
C02550=1125.764,13.483,-50.992,179.652,6.583,149.307
C02551=1125.759,13.732,-51.006,179.653,6.588,149.307
C02552=1125.754,13.982,-51.020,179.655,6.593,149.308
C02553=1125.749,14.232,-51.034,179.655,6.598,149.309
C02554=1125.743,14.481,-51.048,179.656,6.602,149.310
C02555=1125.738,14.731,-51.062,179.657,6.607,149.311
C02556=1125.733,14.981,-51.076,179.658,6.611,149.311
C02557=1125.728,15.230,-51.090,179.658,6.616,149.312
C02558=1125.723,15.479,-51.104,179.659,6.620,149.313
C02559=1125.718,15.729,-51.118,179.661,6.625,149.313
C02560=1125.714,15.979,-51.132,179.662,6.630,149.314
C02561=1125.708,16.228,-51.146,179.663,6.634,149.315
C02562=1125.703,16.478,-51.160,179.663,6.639,149.316
C02563=1125.698,16.728,-51.174,179.664,6.643,149.316
C02564=1125.692,16.977,-51.188,179.665,6.648,149.317
C02565=1125.687,17.226,-51.202,179.666,6.652,149.318
C02566=1125.682,17.476,-51.217,179.667,6.657,149.319
C02567=1125.677,17.726,-51.231,179.668,6.662,149.319
C02568=1125.672,17.975,-51.245,179.669,6.667,149.320
C02569=1125.667,18.225,-51.259,179.670,6.671,149.321
C02570=1125.662,18.474,-51.273,179.671,6.676,149.322
C02571=1125.657,18.724,-51.288,179.672,6.680,149.322
C02572=1125.652,18.974,-51.302,179.673,6.684,149.323
C02573=1125.646,19.223,-51.316,179.674,6.689,149.324
C02574=1125.641,19.472,-51.330,179.674,6.693,149.324
C02575=1125.636,19.722,-51.344,179.675,6.698,149.325
C02576=1125.632,19.972,-51.359,179.677,6.703,149.326
C02577=1125.627,20.222,-51.373,179.678,6.707,149.327
C02578=1125.623,20.436,-51.385,179.679,6.711,149.327
C02579=1125.618,20.652,-51.398,179.680,6.715,149.328
C02580=1125.614,20.866,-51.410,179.680,6.718,149.328
C02581=1125.609,21.082,-51.422,179.681,6.723,149.329
C02582=1125.605,21.297,-51.435,179.682,6.726,149.330
C02583=1125.600,21.512,-51.447,179.683,6.730,149.330
C02584=1125.596,21.727,-51.459,179.683,6.734,149.331
C02585=1125.591,21.942,-51.472,179.685,6.738,149.331
C02586=1125.587,22.192,-51.486,179.686,6.742,149.332
C02587=1125.582,22.441,-51.501,179.687,6.747,149.333
C02588=1125.576,22.690,-51.515,179.687,6.751,149.334
C02589=1125.571,22.940,-51.529,179.688,6.756,149.334
C02590=1125.566,23.190,-51.543,179.689,6.760,149.335
C02591=1125.561,23.440,-51.558,179.690,6.764,149.336
C02592=1125.556,23.689,-51.573,179.691,6.769,149.336
C02593=1125.551,23.939,-51.587,179.693,6.774,149.337
C02594=1125.546,24.188,-51.602,179.694,6.778,149.338
C02595=1125.541,24.437,-51.616,179.695,6.783,149.338
C02596=1125.536,24.686,-51.631,179.696,6.787,149.339
C02597=1125.530,24.936,-51.645,179.697,6.791,149.340
C02598=1125.525,25.186,-51.660,179.698,6.796,149.340
C02599=1125.520,25.436,-51.674,179.699,6.800,149.341
C02600=1125.516,25.685,-51.689,179.700,6.804,149.342
C02601=1125.511,25.935,-51.703,179.701,6.809,149.342
C02602=1125.505,26.185,-51.718,179.702,6.813,149.343
C02603=1125.500,26.434,-51.733,179.703,6.818,149.344
C02604=1125.495,26.683,-51.747,179.704,6.822,149.344
C02605=1125.490,26.933,-51.762,179.705,6.826,149.345
C02606=1125.485,27.181,-51.776,179.706,6.831,149.346
C02607=1125.480,27.432,-51.791,179.707,6.835,149.346
C02608=1125.475,27.681,-51.806,179.708,6.839,149.347
C02609=1125.470,27.930,-51.821,179.709,6.844,149.348
C02610=1125.464,28.180,-51.835,179.711,6.849,149.348
C02611=1125.460,28.429,-51.850,179.712,6.853,149.349
C02612=1125.455,28.679,-51.865,179.713,6.857,149.350
C02613=1125.450,28.929,-51.879,179.714,6.862,149.350
C02614=1125.444,29.178,-51.895,179.715,6.866,149.351
C02615=1125.439,29.428,-51.909,179.716,6.870,149.352
C02616=1125.435,29.677,-51.924,179.717,6.875,149.352
C02617=1125.429,29.927,-51.939,179.718,6.879,149.353
C02618=1125.424,30.176,-51.954,179.719,6.883,149.354
C02619=1125.419,30.426,-51.968,179.720,6.888,149.354
C02620=1125.414,30.675,-51.984,179.721,6.892,149.355
C02621=1125.409,30.925,-51.998,179.722,6.896,149.355
C02622=1125.404,31.174,-52.013,179.723,6.900,149.356
C02623=1125.399,31.424,-52.028,179.724,6.905,149.357
C02624=1125.394,31.673,-52.043,179.725,6.909,149.357
C02625=1125.389,31.922,-52.058,179.726,6.913,149.358
C02626=1125.384,32.172,-52.073,179.728,6.918,149.359
C02627=1125.379,32.421,-52.088,179.729,6.922,149.359
C02628=1125.373,32.671,-52.102,179.730,6.926,149.360
C02629=1125.369,32.921,-52.117,179.731,6.931,149.361
C02630=1125.365,33.170,-52.133,179.732,6.935,149.361
C02631=1125.359,33.420,-52.148,179.733,6.939,149.362
C02632=1125.354,33.669,-52.163,179.734,6.943,149.362
C02633=1125.349,33.919,-52.177,179.735,6.948,149.363
C02634=1125.344,34.134,-52.190,179.737,6.952,149.364
C02635=1125.340,34.349,-52.203,179.737,6.955,149.364
C02636=1125.336,34.564,-52.216,179.739,6.959,149.365
C02637=1125.332,34.780,-52.229,179.739,6.962,149.365
C02638=1125.327,34.995,-52.242,179.740,6.967,149.366
C02639=1125.323,35.209,-52.256,179.741,6.970,149.366
C02640=1125.318,35.424,-52.269,179.742,6.973,149.367
C02641=1125.314,35.640,-52.282,179.743,6.977,149.367
C02642=1125.309,35.889,-52.297,179.744,6.982,149.368
C02643=1125.304,36.139,-52.312,179.746,6.986,149.369
C02644=1125.299,36.388,-52.327,179.747,6.990,149.369
C02645=1125.294,36.637,-52.343,179.748,6.994,149.370
C02646=1125.289,36.887,-52.357,179.749,6.998,149.370
C02647=1125.283,37.136,-52.373,179.750,7.003,149.371
C02648=1125.279,37.385,-52.388,179.751,7.007,149.372
C02649=1125.273,37.635,-52.403,179.752,7.011,149.372
C02650=1125.269,37.885,-52.419,179.754,7.015,149.373
C02651=1125.264,38.135,-52.433,179.755,7.020,149.373
C02652=1125.258,38.384,-52.449,179.756,7.024,149.374
C02653=1125.254,38.633,-52.464,179.757,7.028,149.375
C02654=1125.248,38.882,-52.480,179.758,7.033,149.375
C02655=1125.244,39.132,-52.495,179.760,7.036,149.376
C02656=1125.239,39.382,-52.511,179.761,7.041,149.376
C02657=1125.233,39.631,-52.526,179.762,7.045,149.377
C02658=1125.228,39.881,-52.540,179.763,7.049,149.378
C02659=1125.223,40.130,-52.556,179.765,7.053,149.378
C02660=1125.218,40.379,-52.571,179.766,7.058,149.379
C02661=1125.214,40.629,-52.587,179.767,7.062,149.379
C02662=1125.208,40.879,-52.602,179.768,7.066,149.380
C02663=1125.204,41.128,-52.617,179.769,7.070,149.380
C02664=1125.198,41.377,-52.633,179.770,7.074,149.381
C02665=1125.193,41.627,-52.649,179.771,7.079,149.382
C02666=1125.189,41.876,-52.664,179.773,7.083,149.382
C02667=1125.183,42.126,-52.680,179.774,7.087,149.383
C02668=1125.178,42.375,-52.695,179.775,7.091,149.383
C02669=1125.173,42.624,-52.710,179.777,7.095,149.384
C02670=1125.168,42.874,-52.726,179.778,7.100,149.385
C02671=1125.163,43.124,-52.742,179.779,7.104,149.385
C02672=1125.158,43.373,-52.757,179.780,7.108,149.386
C02673=1125.153,43.622,-52.772,179.781,7.112,149.386
C02674=1125.148,43.872,-52.788,179.783,7.116,149.387
C02675=1125.143,44.122,-52.804,179.784,7.121,149.388
C02676=1125.138,44.371,-52.819,179.785,7.125,149.388
C02677=1125.134,44.620,-52.836,179.786,7.129,149.389
C02678=1125.128,44.870,-52.851,179.788,7.133,149.389
C02679=1125.123,45.119,-52.867,179.789,7.137,149.390
C02680=1125.118,45.369,-52.882,179.789,7.141,149.390
C02681=1125.114,45.618,-52.898,179.791,7.145,149.391
C02682=1125.108,45.868,-52.913,179.792,7.149,149.391
C02683=1125.103,46.117,-52.929,179.793,7.153,149.392
C02684=1125.098,46.367,-52.945,179.795,7.157,149.393
C02685=1125.093,46.616,-52.961,179.796,7.161,149.393
C02686=1125.088,46.865,-52.976,179.797,7.165,149.394
C02687=1125.083,47.115,-52.992,179.798,7.170,149.394
C02688=1125.078,47.365,-53.008,179.799,7.174,149.395
C02689=1125.073,47.614,-53.024,179.801,7.178,149.395
C02690=1125.069,47.829,-53.037,179.802,7.182,149.396
C02691=1125.065,48.044,-53.051,179.803,7.185,149.396
C02692=1125.061,48.259,-53.064,179.804,7.188,149.397
C02693=1125.056,48.473,-53.078,179.805,7.192,149.397
C02694=1125.051,48.689,-53.092,179.806,7.195,149.398
C02695=1125.047,48.904,-53.106,179.807,7.200,149.398
C02696=1125.043,49.118,-53.119,179.808,7.203,149.399
C02697=1125.039,49.334,-53.133,179.810,7.207,149.399
C02698=1125.034,49.583,-53.148,179.810,7.210,149.400
C02699=1125.029,49.833,-53.165,179.812,7.214,149.400
C02700=1125.024,50.082,-53.181,179.813,7.219,149.401
C02701=1125.018,50.331,-53.196,179.815,7.222,149.401
C02702=1125.014,50.581,-53.213,179.816,7.227,149.402
C02703=1125.009,50.830,-53.228,179.817,7.231,149.402
C02704=1125.004,51.080,-53.245,179.818,7.235,149.403
C02705=1124.999,51.329,-53.261,179.820,7.239,149.403
C02706=1124.993,51.579,-53.276,179.821,7.243,149.404
C02707=1124.990,51.828,-53.292,179.822,7.247,149.405
C02708=1124.984,52.077,-53.308,179.824,7.251,149.405
C02709=1124.980,52.327,-53.325,179.825,7.255,149.406
C02710=1124.974,52.576,-53.340,179.826,7.260,149.406
C02711=1124.970,52.826,-53.357,179.828,7.264,149.407
C02712=1124.964,53.075,-53.373,179.829,7.268,149.407
C02713=1124.958,53.325,-53.389,179.830,7.272,149.408
C02714=1124.954,53.574,-53.405,179.832,7.276,149.408
C02715=1124.948,53.824,-53.421,179.833,7.280,149.409
C02716=1124.944,54.073,-53.438,179.834,7.284,149.409
C02717=1124.939,54.322,-53.453,179.836,7.288,149.410
C02718=1124.934,54.572,-53.470,179.837,7.292,149.411
C02719=1124.929,54.821,-53.486,179.838,7.296,149.411
C02720=1124.924,55.071,-53.502,179.839,7.301,149.412
C02721=1124.919,55.320,-53.518,179.840,7.304,149.412
C02722=1124.914,55.570,-53.534,179.842,7.308,149.413
C02723=1124.909,55.819,-53.551,179.843,7.312,149.413
C02724=1124.905,56.069,-53.567,179.845,7.316,149.414
C02725=1124.899,56.317,-53.583,179.846,7.320,149.414
C02726=1124.895,56.567,-53.600,179.847,7.324,149.415
C02727=1124.889,56.817,-53.616,179.848,7.328,149.415
C02728=1124.884,57.066,-53.632,179.850,7.332,149.416
C02729=1124.879,57.315,-53.649,179.851,7.337,149.416
C02730=1124.874,57.565,-53.665,179.853,7.341,149.417
C02731=1124.869,57.814,-53.681,179.854,7.344,149.417
C02732=1124.865,58.063,-53.698,179.855,7.349,149.418
C02733=1124.860,58.313,-53.714,179.857,7.353,149.418
C02734=1124.854,58.562,-53.731,179.858,7.357,149.419
C02735=1124.850,58.812,-53.747,179.859,7.361,149.419
C02736=1124.844,59.061,-53.763,179.861,7.365,149.420
C02737=1124.840,59.311,-53.779,179.862,7.369,149.420
C02738=1124.835,59.560,-53.796,179.864,7.373,149.421
C02739=1124.830,59.809,-53.813,179.865,7.377,149.421
C02740=1124.825,60.060,-53.829,179.866,7.381,149.422
C02741=1124.820,60.308,-53.845,179.867,7.385,149.423
C02742=1124.815,60.558,-53.862,179.868,7.389,149.423
C02743=1124.810,60.807,-53.879,179.870,7.393,149.423
C02744=1124.805,61.056,-53.896,179.871,7.397,149.424
C02745=1124.800,61.306,-53.911,179.873,7.401,149.424
C02746=1124.796,61.521,-53.925,179.874,7.405,149.425
C02747=1124.792,61.736,-53.941,179.875,7.408,149.425
C02748=1124.788,61.950,-53.954,179.876,7.411,149.426
C02749=1124.783,62.165,-53.969,179.878,7.415,149.426
C02750=1124.779,62.380,-53.983,179.879,7.418,149.427
C02751=1124.774,62.595,-53.997,179.880,7.422,149.427
C02752=1124.771,62.810,-54.011,179.881,7.425,149.427
C02753=1124.766,63.025,-54.026,179.883,7.429,149.428
C02754=1124.761,63.274,-54.042,179.883,7.432,149.429
C02755=1124.756,63.524,-54.060,179.885,7.436,149.429
C02756=1124.751,63.773,-54.076,179.886,7.440,149.429
C02757=1124.746,64.022,-54.093,179.887,7.444,149.430
C02758=1124.741,64.272,-54.110,179.889,7.448,149.430
C02759=1124.737,64.521,-54.127,179.891,7.452,149.431
C02760=1124.732,64.770,-54.143,179.892,7.457,149.432
C02761=1124.726,65.020,-54.160,179.893,7.460,149.432
C02762=1124.722,65.269,-54.177,179.895,7.464,149.432
C02763=1124.717,65.518,-54.193,179.896,7.469,149.433
C02764=1124.712,65.768,-54.210,179.897,7.473,149.433
C02765=1124.707,66.018,-54.227,179.899,7.476,149.434
C02766=1124.701,66.267,-54.244,179.900,7.481,149.435
C02767=1124.697,66.516,-54.261,179.902,7.485,149.435
C02768=1124.692,66.766,-54.277,179.903,7.489,149.435
C02769=1124.687,67.015,-54.294,179.904,7.493,149.436
C02770=1124.682,67.264,-54.311,179.906,7.497,149.436
C02771=1124.677,67.514,-54.328,179.908,7.501,149.437
C02772=1124.672,67.763,-54.345,179.909,7.505,149.438
C02773=1124.667,68.013,-54.362,179.910,7.509,149.438
C02774=1124.662,68.261,-54.379,179.911,7.512,149.438
C02775=1124.658,68.511,-54.396,179.913,7.516,149.439
C02776=1124.653,68.761,-54.413,179.914,7.520,149.439
C02777=1124.648,69.010,-54.430,179.915,7.524,149.440
C02778=1124.642,69.259,-54.447,179.917,7.528,149.440
C02779=1124.638,69.509,-54.463,179.918,7.532,149.441
C02780=1124.633,69.758,-54.481,179.920,7.536,149.441
C02781=1124.628,70.007,-54.498,179.921,7.540,149.442
C02782=1124.623,70.257,-54.515,179.923,7.544,149.442
C02783=1124.618,70.506,-54.531,179.924,7.548,149.443
C02784=1124.613,70.756,-54.549,179.926,7.552,149.443
C02785=1124.608,71.005,-54.567,179.927,7.556,149.444
C02786=1124.604,71.254,-54.583,179.928,7.560,149.444
C02787=1124.598,71.504,-54.601,179.930,7.564,149.445
C02788=1124.593,71.753,-54.617,179.931,7.568,149.445
C02789=1124.588,72.002,-54.635,179.933,7.572,149.446
C02790=1124.584,72.252,-54.652,179.934,7.576,149.446
C02791=1124.579,72.501,-54.669,179.936,7.580,149.447
C02792=1124.574,72.751,-54.687,179.937,7.584,149.447
C02793=1124.569,73.000,-54.703,179.939,7.588,149.448
C02794=1124.563,73.249,-54.720,179.940,7.592,149.448
C02795=1124.559,73.498,-54.738,179.941,7.596,149.449
C02796=1124.554,73.748,-54.755,179.943,7.600,149.449
C02797=1124.549,73.998,-54.772,179.944,7.603,149.450
C02798=1124.545,74.247,-54.790,179.945,7.608,149.450
C02799=1124.539,74.496,-54.807,179.947,7.611,149.451
C02800=1124.535,74.746,-54.825,179.948,7.615,149.451
C02801=1124.530,74.995,-54.842,179.950,7.619,149.451
C02802=1124.525,75.209,-54.857,179.951,7.623,149.452
C02803=1124.521,75.424,-54.871,179.952,7.626,149.452
C02804=1124.517,75.639,-54.887,179.954,7.630,149.453
C02805=1124.513,75.854,-54.902,179.955,7.633,149.453
C02806=1124.509,76.069,-54.916,179.956,7.636,149.454
C02807=1124.505,76.284,-54.931,179.957,7.640,149.454
C02808=1124.500,76.498,-54.946,179.958,7.643,149.454
C02809=1124.496,76.713,-54.961,179.960,7.647,149.455
C02810=1124.491,76.962,-54.979,179.961,7.650,149.455
C02811=1124.486,77.212,-54.996,179.961,7.654,149.456
C02812=1124.481,77.461,-55.014,179.963,7.658,149.457
C02813=1124.476,77.711,-55.031,179.964,7.661,149.457
C02814=1124.471,77.960,-55.049,179.965,7.666,149.458
C02815=1124.467,78.209,-55.066,179.966,7.669,149.458
C02816=1124.462,78.458,-55.084,179.967,7.673,149.459
C02817=1124.457,78.708,-55.102,179.968,7.676,149.459
C02818=1124.452,78.957,-55.119,179.969,7.680,149.460
C02819=1124.447,79.207,-55.137,179.970,7.684,149.460
C02820=1124.442,79.456,-55.154,179.971,7.688,149.461
C02821=1124.437,79.705,-55.172,179.971,7.691,149.462
C02822=1124.432,79.954,-55.190,179.973,7.695,149.462
C02823=1124.427,80.204,-55.207,179.974,7.699,149.463
C02824=1124.422,80.453,-55.224,179.975,7.703,149.463
C02825=1124.418,80.702,-55.242,179.976,7.707,149.464
C02826=1124.412,80.951,-55.259,179.977,7.710,149.464
C02827=1124.407,81.200,-55.277,179.978,7.714,149.465
C02828=1124.403,81.450,-55.295,179.979,7.717,149.465
C02829=1124.397,81.699,-55.312,179.981,7.721,149.466
C02830=1124.392,81.949,-55.330,179.981,7.725,149.466
C02831=1124.389,82.198,-55.348,179.983,7.729,149.467
C02832=1124.384,82.448,-55.365,179.984,7.733,149.467
C02833=1124.379,82.697,-55.383,179.985,7.736,149.468
C02834=1124.374,82.946,-55.401,179.986,7.740,149.468
C02835=1124.369,83.196,-55.419,179.988,7.744,149.469
C02836=1124.364,83.445,-55.436,179.988,7.748,149.469
C02837=1124.359,83.695,-55.454,179.990,7.752,149.470
C02838=1124.354,83.944,-55.472,179.991,7.756,149.470
C02839=1124.349,84.193,-55.490,179.992,7.759,149.471
C02840=1124.344,84.443,-55.508,179.994,7.763,149.471
C02841=1124.340,84.692,-55.525,179.995,7.767,149.472
C02842=1124.335,84.941,-55.543,179.996,7.771,149.472
C02843=1124.330,85.190,-55.561,179.997,7.774,149.473
C02844=1124.325,85.439,-55.579,179.998,7.779,149.474
C02845=1124.320,85.688,-55.597,-180.000,7.782,149.474
C02846=1124.315,85.938,-55.614,-179.998,7.786,149.474
C02847=1124.310,86.187,-55.632,-179.998,7.790,149.475
C02848=1124.305,86.436,-55.650,-179.996,7.794,149.475
C02849=1124.301,86.686,-55.669,-179.995,7.798,149.476
C02850=1124.296,86.935,-55.687,-179.993,7.802,149.476
C02851=1124.291,87.185,-55.705,-179.992,7.806,149.477
C02852=1124.286,87.434,-55.723,-179.991,7.809,149.477
C02853=1124.281,87.683,-55.740,-179.989,7.813,149.478
C02854=1124.276,87.932,-55.758,-179.988,7.817,149.478
C02855=1124.271,88.181,-55.776,-179.987,7.821,149.479
C02856=1124.266,88.430,-55.794,-179.985,7.825,149.479
C02857=1124.262,88.680,-55.813,-179.983,7.829,149.480
C02858=1124.257,88.894,-55.828,-179.983,7.832,149.480
C02859=1124.252,89.109,-55.844,-179.982,7.835,149.481
C02860=1124.248,89.324,-55.859,-179.980,7.839,149.481
C02861=1124.244,89.539,-55.875,-179.979,7.842,149.481
C02862=1124.240,89.754,-55.890,-179.978,7.845,149.482
C02863=1124.236,89.969,-55.906,-179.976,7.849,149.482
C02864=1124.233,90.183,-55.922,-179.975,7.852,149.483
C02865=1124.228,90.398,-55.938,-179.974,7.855,149.483
C02866=1124.223,90.647,-55.956,-179.972,7.859,149.483
C02867=1124.218,90.897,-55.974,-179.971,7.863,149.484
C02868=1124.213,91.146,-55.992,-179.970,7.867,149.484
C02869=1124.208,91.395,-56.010,-179.968,7.871,149.485
C02870=1124.203,91.644,-56.028,-179.967,7.875,149.485
C02871=1124.199,91.894,-56.046,-179.965,7.879,149.486
C02872=1124.194,92.143,-56.064,-179.963,7.882,149.486
C02873=1124.188,92.393,-56.083,-179.962,7.886,149.487
C02874=1124.184,92.641,-56.101,-179.960,7.890,149.487
C02875=1124.179,92.891,-56.120,-179.959,7.894,149.487
C02876=1124.174,93.140,-56.138,-179.957,7.898,149.488
C02877=1124.169,93.389,-56.156,-179.955,7.902,149.488
C02878=1124.165,93.639,-56.174,-179.954,7.906,149.489
C02879=1124.159,93.887,-56.193,-179.952,7.910,149.489
C02880=1124.155,94.137,-56.211,-179.951,7.914,149.490
C02881=1124.150,94.386,-56.229,-179.949,7.917,149.490
C02882=1124.145,94.636,-56.247,-179.947,7.921,149.490
C02883=1124.139,94.885,-56.266,-179.946,7.925,149.491
C02884=1124.135,95.134,-56.285,-179.944,7.929,149.491
C02885=1124.131,95.384,-56.303,-179.942,7.934,149.492
C02886=1124.126,95.633,-56.321,-179.940,7.938,149.492
C02887=1124.121,95.882,-56.340,-179.938,7.941,149.492
C02888=1124.116,96.131,-56.358,-179.937,7.945,149.493
C02889=1124.111,96.381,-56.376,-179.935,7.949,149.493
C02890=1124.106,96.629,-56.395,-179.933,7.953,149.494
C02891=1124.101,96.879,-56.414,-179.932,7.957,149.494
C02892=1124.096,97.129,-56.432,-179.930,7.961,149.495
C02893=1124.092,97.377,-56.451,-179.928,7.964,149.495
C02894=1124.087,97.627,-56.470,-179.926,7.969,149.495
C02895=1124.082,97.876,-56.488,-179.924,7.973,149.496
C02896=1124.077,98.125,-56.506,-179.923,7.977,149.496
C02897=1124.072,98.375,-56.525,-179.921,7.981,149.497
C02898=1124.068,98.624,-56.544,-179.919,7.984,149.497
C02899=1124.063,98.873,-56.562,-179.918,7.988,149.497
C02900=1124.058,99.123,-56.582,-179.915,7.993,149.498
C02901=1124.053,99.372,-56.600,-179.913,7.996,149.498
C02902=1124.048,99.621,-56.619,-179.912,8.000,149.498
C02903=1124.043,99.870,-56.637,-179.910,8.004,149.499
C02904=1124.039,100.119,-56.656,-179.908,8.007,149.499
C02905=1124.034,100.369,-56.675,-179.906,8.012,149.499
C02906=1124.029,100.618,-56.693,-179.904,8.016,149.500
C02907=1124.024,100.867,-56.712,-179.902,8.019,149.500
C02908=1124.020,101.116,-56.731,-179.900,8.023,149.500
C02909=1124.014,101.366,-56.750,-179.898,8.028,149.501
C02910=1124.009,101.615,-56.768,-179.896,8.031,149.501
C02911=1124.005,101.864,-56.787,-179.894,8.035,149.501
C02912=1124.000,102.113,-56.806,-179.892,8.040,149.502
C02913=1123.996,102.363,-56.825,-179.890,8.043,149.502
C02914=1123.991,102.578,-56.841,-179.888,8.047,149.502
C02915=1123.987,102.792,-56.857,-179.887,8.050,149.503
C02916=1123.982,103.006,-56.874,-179.885,8.053,149.503
C02917=1123.979,103.221,-56.890,-179.883,8.057,149.503
C02918=1123.974,103.436,-56.906,-179.882,8.060,149.503
C02919=1123.970,103.650,-56.922,-179.880,8.063,149.504
C02920=1123.966,103.864,-56.939,-179.878,8.067,149.504
C02921=1123.961,104.079,-56.956,-179.876,8.070,149.504
C02922=1123.957,104.329,-56.974,-179.874,8.074,149.505
C02923=1123.952,104.578,-56.993,-179.872,8.078,149.505
C02924=1123.948,104.827,-57.012,-179.869,8.082,149.505
C02925=1123.942,105.076,-57.032,-179.868,8.086,149.505
C02926=1123.938,105.326,-57.050,-179.866,8.089,149.506
C02927=1123.933,105.574,-57.069,-179.863,8.094,149.506
C02928=1123.928,105.824,-57.089,-179.861,8.098,149.506
C02929=1123.923,106.073,-57.108,-179.859,8.101,149.506
C02930=1123.919,106.322,-57.127,-179.856,8.105,149.507
C02931=1123.914,106.571,-57.145,-179.854,8.109,149.507
C02932=1123.909,106.821,-57.165,-179.852,8.114,149.507
C02933=1123.904,107.070,-57.184,-179.850,8.117,149.508
C02934=1123.900,107.319,-57.203,-179.848,8.121,149.508
C02935=1123.895,107.569,-57.223,-179.845,8.125,149.508
C02936=1123.889,107.817,-57.242,-179.843,8.128,149.508
C02937=1123.885,108.067,-57.261,-179.841,8.133,149.508
C02938=1123.880,108.316,-57.281,-179.839,8.136,149.509
C02939=1123.875,108.565,-57.300,-179.836,8.141,149.509
C02940=1123.870,108.815,-57.319,-179.834,8.144,149.509
C02941=1123.866,109.064,-57.338,-179.832,8.149,149.510
C02942=1123.861,109.313,-57.358,-179.830,8.152,149.510
C02943=1123.856,109.562,-57.377,-179.827,8.156,149.510
C02944=1123.852,109.812,-57.396,-179.825,8.160,149.510
C02945=1123.846,110.060,-57.415,-179.823,8.163,149.510
C02946=1123.842,110.309,-57.436,-179.820,8.168,149.511
C02947=1123.837,110.559,-57.455,-179.818,8.171,149.511
C02948=1123.832,110.808,-57.475,-179.815,8.175,149.511
C02949=1123.828,111.057,-57.494,-179.813,8.179,149.511
C02950=1123.822,111.306,-57.513,-179.811,8.182,149.512
C02951=1123.818,111.556,-57.533,-179.809,8.186,149.512
C02952=1123.813,111.805,-57.552,-179.807,8.189,149.512
C02953=1123.808,112.054,-57.572,-179.805,8.193,149.512
C02954=1123.803,112.304,-57.591,-179.803,8.197,149.513
C02955=1123.799,112.553,-57.610,-179.801,8.200,149.513
C02956=1123.794,112.801,-57.630,-179.799,8.204,149.513
C02957=1123.789,113.051,-57.650,-179.798,8.207,149.513
C02958=1123.784,113.300,-57.670,-179.796,8.210,149.514
C02959=1123.779,113.549,-57.689,-179.794,8.214,149.514
C02960=1123.774,113.799,-57.709,-179.792,8.217,149.514
C02961=1123.770,114.048,-57.729,-179.790,8.221,149.514
C02962=1123.764,114.296,-57.748,-179.788,8.225,149.515
C02963=1123.760,114.546,-57.767,-179.786,8.228,149.515
C02964=1123.756,114.795,-57.787,-179.784,8.232,149.515
C02965=1123.751,115.044,-57.807,-179.783,8.234,149.515
C02966=1123.746,115.293,-57.827,-179.781,8.238,149.516
C02967=1123.741,115.543,-57.846,-179.779,8.242,149.516
C02968=1123.736,115.792,-57.866,-179.777,8.245,149.516
C02969=1123.731,116.040,-57.886,-179.775,8.249,149.517
C02970=1123.727,116.256,-57.903,-179.774,8.252,149.517
C02971=1123.723,116.470,-57.920,-179.772,8.254,149.517
C02972=1123.719,116.685,-57.937,-179.770,8.258,149.517
C02973=1123.715,116.899,-57.954,-179.769,8.261,149.517
C02974=1123.711,117.114,-57.971,-179.767,8.263,149.518
C02975=1123.707,117.328,-57.988,-179.766,8.267,149.518
C02976=1123.703,117.543,-58.005,-179.764,8.270,149.518
C02977=1123.699,117.756,-58.022,-179.763,8.273,149.519
C02978=1123.694,118.006,-58.042,-179.761,8.276,149.519
C02979=1123.689,118.256,-58.062,-179.759,8.280,149.519
C02980=1123.684,118.504,-58.082,-179.757,8.283,149.519
C02981=1123.680,118.753,-58.101,-179.755,8.286,149.519
C02982=1123.675,119.002,-58.122,-179.754,8.290,149.520
C02983=1123.670,119.252,-58.142,-179.751,8.293,149.520
C02984=1123.665,119.500,-58.162,-179.749,8.297,149.520
C02985=1123.660,119.750,-58.182,-179.747,8.300,149.521
C02986=1123.656,119.999,-58.202,-179.746,8.303,149.521
C02987=1123.651,120.249,-58.222,-179.744,8.307,149.521
C02988=1123.646,120.497,-58.242,-179.742,8.310,149.521
C02989=1123.642,120.747,-58.262,-179.740,8.314,149.522
C02990=1123.637,120.995,-58.282,-179.739,8.316,149.522
C02991=1123.632,121.245,-58.301,-179.737,8.320,149.522
C02992=1123.627,121.494,-58.322,-179.735,8.324,149.523
C02993=1123.623,121.743,-58.342,-179.733,8.327,149.523
C02994=1123.618,121.993,-58.362,-179.731,8.330,149.523
C02995=1123.613,122.242,-58.383,-179.729,8.334,149.523
C02996=1123.608,122.491,-58.402,-179.728,8.337,149.524
C02997=1123.603,122.739,-58.423,-179.726,8.341,149.524
C02998=1123.599,122.989,-58.442,-179.724,8.344,149.524
C02999=1123.594,123.238,-58.463,-179.722,8.347,149.524
C03000=1123.589,123.487,-58.483,-179.720,8.351,149.525
C03001=1123.584,123.737,-58.503,-179.719,8.354,149.525
C03002=1123.580,123.986,-58.524,-179.717,8.357,149.525
C03003=1123.575,124.235,-58.544,-179.715,8.361,149.525
C03004=1123.571,124.484,-58.564,-179.713,8.364,149.526
C03005=1123.565,124.734,-58.585,-179.712,8.367,149.526
C03006=1123.560,124.982,-58.605,-179.710,8.371,149.526
C03007=1123.556,125.231,-58.625,-179.708,8.374,149.527
C03008=1123.551,125.480,-58.645,-179.706,8.377,149.527
C03009=1123.547,125.729,-58.665,-179.705,8.381,149.527
C03010=1123.542,125.978,-58.686,-179.703,8.384,149.527
C03011=1123.537,126.227,-58.706,-179.701,8.388,149.528
C03012=1123.532,126.477,-58.726,-179.699,8.391,149.528
C03013=1123.527,126.726,-58.747,-179.697,8.394,149.528
C03014=1123.523,126.975,-58.767,-179.695,8.398,149.529
C03015=1123.518,127.224,-58.788,-179.694,8.401,149.529
C03016=1123.514,127.473,-58.808,-179.692,8.404,149.529
C03017=1123.509,127.722,-58.829,-179.690,8.408,149.529
C03018=1123.504,127.972,-58.849,-179.689,8.411,149.530
C03019=1123.500,128.221,-58.869,-179.687,8.414,149.530
C03020=1123.494,128.470,-58.890,-179.685,8.418,149.530
C03021=1123.490,128.719,-58.910,-179.683,8.420,149.530
C03022=1123.486,128.968,-58.931,-179.682,8.424,149.531
C03023=1123.480,129.217,-58.952,-179.680,8.428,149.531
C03024=1123.476,129.466,-58.972,-179.678,8.431,149.531
C03025=1123.471,129.715,-58.993,-179.677,8.434,149.532
C03026=1123.466,129.929,-59.010,-179.675,8.437,149.532
C03027=1123.463,130.144,-59.027,-179.674,8.440,149.532
C03028=1123.459,130.359,-59.045,-179.672,8.443,149.532
C03029=1123.455,130.573,-59.063,-179.671,8.445,149.533
C03030=1123.450,130.788,-59.081,-179.669,8.448,149.533
C03031=1123.447,131.002,-59.099,-179.667,8.451,149.533
C03032=1123.442,131.216,-59.116,-179.666,8.454,149.533
C03033=1123.439,131.430,-59.134,-179.664,8.457,149.533
C03034=1123.433,131.680,-59.155,-179.663,8.460,149.534
C03035=1123.429,131.929,-59.175,-179.661,8.463,149.534
C03036=1123.424,132.178,-59.196,-179.659,8.467,149.534
C03037=1123.419,132.427,-59.217,-179.658,8.470,149.535
C03038=1123.414,132.676,-59.238,-179.656,8.474,149.535
C03039=1123.410,132.925,-59.258,-179.654,8.477,149.535
C03040=1123.405,133.174,-59.279,-179.653,8.480,149.536
C03041=1123.400,133.423,-59.299,-179.651,8.484,149.536
C03042=1123.395,133.672,-59.320,-179.650,8.486,149.536
C03043=1123.391,133.921,-59.341,-179.648,8.490,149.537
C03044=1123.386,134.170,-59.362,-179.646,8.494,149.537
C03045=1123.382,134.420,-59.383,-179.644,8.496,149.537
C03046=1123.377,134.669,-59.404,-179.643,8.500,149.537
C03047=1123.372,134.918,-59.424,-179.641,8.503,149.538
C03048=1123.367,135.167,-59.445,-179.639,8.507,149.538
C03049=1123.363,135.416,-59.466,-179.638,8.510,149.538
C03050=1123.358,135.665,-59.487,-179.636,8.513,149.539
C03051=1123.353,135.914,-59.508,-179.635,8.517,149.539
C03052=1123.348,136.163,-59.529,-179.633,8.520,149.539
C03053=1123.344,136.412,-59.549,-179.631,8.523,149.539
C03054=1123.339,136.662,-59.571,-179.630,8.526,149.540
C03055=1123.334,136.910,-59.592,-179.628,8.530,149.540
C03056=1123.330,137.159,-59.613,-179.627,8.533,149.540
C03057=1123.325,137.409,-59.634,-179.625,8.536,149.541
C03058=1123.320,137.658,-59.654,-179.623,8.540,149.541
C03059=1123.315,137.906,-59.676,-179.622,8.543,149.541
C03060=1123.310,138.155,-59.697,-179.620,8.546,149.542
C03061=1123.306,138.405,-59.717,-179.619,8.550,149.542
C03062=1123.302,138.654,-59.739,-179.617,8.553,149.542
C03063=1123.297,138.903,-59.759,-179.616,8.556,149.543
C03064=1123.292,139.152,-59.780,-179.614,8.560,149.543
C03065=1123.287,139.401,-59.802,-179.611,8.563,149.543
C03066=1123.283,139.650,-59.822,-179.610,8.566,149.544
C03067=1123.278,139.900,-59.844,-179.608,8.570,149.544
C03068=1123.273,140.148,-59.865,-179.607,8.573,149.544
C03069=1123.269,140.397,-59.886,-179.605,8.576,149.544
C03070=1123.264,140.646,-59.907,-179.604,8.579,149.545
C03071=1123.259,140.896,-59.929,-179.602,8.583,149.545
C03072=1123.255,141.145,-59.949,-179.601,8.586,149.546
C03073=1123.250,141.393,-59.971,-179.599,8.589,149.546
C03074=1123.245,141.643,-59.992,-179.598,8.592,149.546
C03075=1123.240,141.891,-60.013,-179.596,8.596,149.546
C03076=1123.236,142.141,-60.034,-179.595,8.599,149.547
C03077=1123.231,142.390,-60.055,-179.593,8.603,149.547
C03078=1123.226,142.639,-60.077,-179.592,8.606,149.548
C03079=1123.222,142.888,-60.097,-179.590,8.610,149.548
C03080=1123.217,143.137,-60.119,-179.588,8.613,149.548
C03081=1123.212,143.386,-60.140,-179.587,8.616,149.549
C03082=1123.209,143.600,-60.159,-179.586,8.619,149.549
C03083=1123.204,143.815,-60.177,-179.585,8.622,149.549
C03084=1123.200,144.028,-60.196,-179.583,8.625,149.550
C03085=1123.196,144.243,-60.214,-179.582,8.627,149.550
C03086=1123.192,144.457,-60.233,-179.581,8.630,149.550
C03087=1123.188,144.672,-60.250,-179.579,8.633,149.550
C03088=1123.184,144.886,-60.269,-179.578,8.636,149.551
C03089=1123.181,145.100,-60.287,-179.577,8.639,149.551
C03090=1123.175,145.350,-60.308,-179.574,8.643,149.551
C03091=1123.171,145.598,-60.330,-179.572,8.647,149.552
C03092=1123.166,145.847,-60.352,-179.569,8.651,149.552
C03093=1123.161,146.097,-60.373,-179.567,8.655,149.552
C03094=1123.156,146.345,-60.395,-179.564,8.658,149.552
C03095=1123.152,146.594,-60.416,-179.561,8.663,149.552
C03096=1123.148,146.844,-60.437,-179.559,8.666,149.553
C03097=1123.143,147.092,-60.459,-179.557,8.670,149.553
C03098=1123.138,147.341,-60.480,-179.555,8.674,149.553
C03099=1123.133,147.591,-60.502,-179.552,8.678,149.553
C03100=1123.128,147.840,-60.523,-179.549,8.681,149.553
C03101=1123.124,148.088,-60.545,-179.547,8.685,149.554
C03102=1123.119,148.338,-60.567,-179.545,8.689,149.554
C03103=1123.114,148.587,-60.588,-179.542,8.693,149.554
C03104=1123.109,148.836,-60.610,-179.540,8.697,149.554
C03105=1123.105,149.085,-60.632,-179.537,8.701,149.554
C03106=1123.100,149.334,-60.654,-179.535,8.704,149.554
C03107=1123.096,149.583,-60.676,-179.532,8.708,149.555
C03108=1123.091,149.832,-60.697,-179.530,8.712,149.555
C03109=1123.086,150.081,-60.718,-179.527,8.715,149.555
C03110=1123.081,150.330,-60.740,-179.525,8.719,149.555
C03111=1123.077,150.579,-60.762,-179.522,8.723,149.555
C03112=1123.072,150.828,-60.784,-179.520,8.726,149.555
C03113=1123.067,151.077,-60.806,-179.517,8.730,149.556
C03114=1123.063,151.325,-60.827,-179.515,8.734,149.556
C03115=1123.058,151.575,-60.849,-179.513,8.737,149.556
C03116=1123.053,151.823,-60.871,-179.510,8.741,149.556
C03117=1123.049,152.073,-60.893,-179.508,8.744,149.556
C03118=1123.044,152.321,-60.915,-179.505,8.748,149.556
C03119=1123.040,152.571,-60.937,-179.503,8.752,149.557
C03120=1123.035,152.819,-60.959,-179.500,8.755,149.557
C03121=1123.031,153.069,-60.981,-179.498,8.758,149.557
C03122=1123.026,153.317,-61.002,-179.495,8.763,149.557
C03123=1123.021,153.567,-61.025,-179.493,8.766,149.557
C03124=1123.016,153.816,-61.047,-179.491,8.769,149.557
C03125=1123.012,154.065,-61.069,-179.488,8.772,149.558
C03126=1123.007,154.314,-61.090,-179.485,8.777,149.558
C03127=1123.003,154.563,-61.112,-179.483,8.780,149.558
C03128=1122.998,154.812,-61.134,-179.481,8.783,149.558
C03129=1122.993,155.061,-61.157,-179.478,8.786,149.558
C03130=1122.988,155.310,-61.178,-179.476,8.791,149.558
C03131=1122.984,155.559,-61.201,-179.473,8.794,149.558
C03132=1122.979,155.807,-61.223,-179.471,8.797,149.559
C03133=1122.975,156.057,-61.245,-179.468,8.800,149.559
C03134=1122.969,156.305,-61.267,-179.466,8.804,149.559
C03135=1122.965,156.555,-61.289,-179.463,8.808,149.559
C03136=1122.960,156.803,-61.311,-179.461,8.811,149.559
C03137=1122.956,157.052,-61.334,-179.459,8.814,149.559
C03138=1122.952,157.266,-61.353,-179.457,8.817,149.559
C03139=1122.948,157.481,-61.372,-179.455,8.820,149.559
C03140=1122.944,157.695,-61.391,-179.452,8.823,149.559
C03141=1122.940,157.909,-61.410,-179.451,8.826,149.560
C03142=1122.936,158.123,-61.429,-179.448,8.829,149.560
C03143=1122.932,158.337,-61.448,-179.447,8.832,149.560
C03144=1122.928,158.552,-61.467,-179.444,8.835,149.560
C03145=1122.924,158.766,-61.486,-179.442,8.837,149.560
C03146=1122.920,159.014,-61.509,-179.440,8.841,149.560
C03147=1122.915,159.264,-61.532,-179.437,8.845,149.560
C03148=1122.910,159.513,-61.554,-179.435,8.848,149.560
C03149=1122.906,159.761,-61.576,-179.432,8.851,149.560
C03150=1122.901,160.011,-61.599,-179.430,8.854,149.561
C03151=1122.896,160.259,-61.621,-179.428,8.858,149.561
C03152=1122.892,160.508,-61.643,-179.425,8.861,149.561
C03153=1122.887,160.758,-61.666,-179.423,8.864,149.561
C03154=1122.882,161.006,-61.688,-179.421,8.867,149.561
C03155=1122.878,161.255,-61.710,-179.418,8.871,149.561
C03156=1122.873,161.504,-61.734,-179.416,8.874,149.561
C03157=1122.869,161.753,-61.756,-179.414,8.877,149.561
C03158=1122.864,162.002,-61.779,-179.411,8.880,149.561
C03159=1122.860,162.252,-61.801,-179.409,8.884,149.562
C03160=1122.855,162.500,-61.823,-179.406,8.887,149.562
C03161=1122.850,162.749,-61.846,-179.404,8.890,149.562
C03162=1122.846,162.998,-61.869,-179.402,8.893,149.562
C03163=1122.840,163.247,-61.891,-179.399,8.897,149.562
C03164=1122.836,163.496,-61.914,-179.397,8.900,149.562
C03165=1122.832,163.745,-61.937,-179.395,8.903,149.562
C03166=1122.827,163.994,-61.959,-179.392,8.906,149.562
C03167=1122.822,164.242,-61.982,-179.390,8.909,149.562
C03168=1122.818,164.492,-62.004,-179.388,8.913,149.563
C03169=1122.813,164.741,-62.028,-179.385,8.916,149.563
C03170=1122.809,164.989,-62.050,-179.383,8.918,149.563
C03171=1122.804,165.238,-62.073,-179.381,8.922,149.563
C03172=1122.800,165.487,-62.095,-179.379,8.925,149.563
C03173=1122.795,165.736,-62.119,-179.376,8.928,149.563
C03174=1122.790,165.985,-62.140,-179.374,8.931,149.563
C03175=1122.785,166.234,-62.164,-179.371,8.935,149.563
C03176=1122.781,166.483,-62.187,-179.369,8.938,149.563
C03177=1122.776,166.732,-62.209,-179.366,8.941,149.563
C03178=1122.772,166.981,-62.233,-179.364,8.944,149.563
C03179=1122.767,167.229,-62.255,-179.362,8.947,149.564
C03180=1122.762,167.478,-62.278,-179.360,8.950,149.564
C03181=1122.757,167.728,-62.301,-179.358,8.953,149.564
C03182=1122.754,167.977,-62.324,-179.355,8.956,149.564
C03183=1122.749,168.226,-62.347,-179.353,8.959,149.564
C03184=1122.744,168.474,-62.369,-179.350,8.962,149.564
C03185=1122.740,168.723,-62.393,-179.348,8.966,149.564
C03186=1122.735,168.972,-62.416,-179.346,8.968,149.564
C03187=1122.731,169.221,-62.438,-179.344,8.971,149.564
C03188=1122.726,169.470,-62.462,-179.342,8.975,149.564
C03189=1122.721,169.718,-62.485,-179.339,8.978,149.564
C03190=1122.717,169.967,-62.507,-179.337,8.981,149.565
C03191=1122.712,170.216,-62.531,-179.335,8.983,149.565
C03192=1122.707,170.465,-62.554,-179.333,8.987,149.565
C03193=1122.703,170.714,-62.577,-179.330,8.990,149.565
C03194=1122.698,170.928,-62.597,-179.328,8.992,149.565
C03195=1122.695,171.142,-62.616,-179.326,8.995,149.565
C03196=1122.691,171.357,-62.637,-179.324,8.998,149.565
C03197=1122.687,171.571,-62.656,-179.322,9.001,149.565
C03198=1122.683,171.784,-62.676,-179.320,9.003,149.565
C03199=1122.679,171.999,-62.697,-179.319,9.005,149.565
C03200=1122.675,172.212,-62.717,-179.316,9.009,149.565
C03201=1122.671,172.427,-62.736,-179.315,9.011,149.565
C03202=1122.666,172.676,-62.759,-179.313,9.013,149.565
C03203=1122.662,172.925,-62.782,-179.311,9.017,149.566
C03204=1122.657,173.174,-62.806,-179.308,9.020,149.566
C03205=1122.653,173.422,-62.828,-179.306,9.023,149.566
C03206=1122.649,173.671,-62.853,-179.304,9.025,149.566
C03207=1122.644,173.920,-62.876,-179.302,9.029,149.566
C03208=1122.639,174.169,-62.899,-179.299,9.032,149.566
C03209=1122.634,174.417,-62.922,-179.297,9.034,149.566
C03210=1122.630,174.666,-62.945,-179.295,9.038,149.566
C03211=1122.625,174.915,-62.968,-179.292,9.041,149.566
C03212=1122.621,175.164,-62.992,-179.291,9.043,149.566
C03213=1122.616,175.413,-63.015,-179.288,9.046,149.567
C03214=1122.611,175.661,-63.039,-179.286,9.050,149.567
C03215=1122.607,175.911,-63.063,-179.284,9.052,149.567
C03216=1122.602,176.160,-63.086,-179.282,9.055,149.567
C03217=1122.597,176.409,-63.109,-179.279,9.059,149.567
C03218=1122.593,176.657,-63.132,-179.278,9.061,149.567
C03219=1122.589,176.906,-63.155,-179.275,9.064,149.567
C03220=1122.584,177.155,-63.179,-179.273,9.068,149.567
C03221=1122.580,177.404,-63.203,-179.271,9.070,149.567
C03222=1122.575,177.653,-63.226,-179.269,9.073,149.567
C03223=1122.570,177.902,-63.250,-179.266,9.077,149.568
C03224=1122.566,178.150,-63.274,-179.265,9.079,149.568
C03225=1122.561,178.399,-63.297,-179.262,9.082,149.568
C03226=1122.556,178.648,-63.320,-179.261,9.085,149.568
C03227=1122.552,178.897,-63.344,-179.258,9.088,149.568
C03228=1122.547,179.146,-63.368,-179.256,9.091,149.568
C03229=1122.543,179.395,-63.391,-179.253,9.094,149.568
C03230=1122.538,179.643,-63.415,-179.250,9.097,149.568
C03231=1122.534,179.892,-63.439,-179.248,9.100,149.568
C03232=1122.529,180.141,-63.462,-179.245,9.104,149.568
C03233=1122.525,180.390,-63.486,-179.242,9.107,149.568
C03234=1122.520,180.639,-63.510,-179.240,9.110,149.568
C03235=1122.516,180.888,-63.534,-179.237,9.114,149.568
C03236=1122.511,181.137,-63.557,-179.234,9.117,149.568
C03237=1122.507,181.385,-63.581,-179.231,9.120,149.568
C03238=1122.502,181.634,-63.605,-179.229,9.123,149.568
C03239=1122.497,181.883,-63.628,-179.225,9.127,149.568
C03240=1122.493,182.132,-63.652,-179.223,9.130,149.568
C03241=1122.488,182.381,-63.675,-179.220,9.133,149.568
C03242=1122.484,182.629,-63.699,-179.217,9.136,149.568
C03243=1122.479,182.878,-63.723,-179.215,9.139,149.568
C03244=1122.476,183.127,-63.747,-179.212,9.142,149.568
C03245=1122.471,183.376,-63.771,-179.210,9.145,149.568
C03246=1122.466,183.625,-63.795,-179.207,9.148,149.568
C03247=1122.461,183.874,-63.819,-179.204,9.151,149.568
C03248=1122.457,184.123,-63.843,-179.202,9.154,149.568
C03249=1122.452,184.371,-63.867,-179.199,9.157,149.568
C03250=1122.448,184.586,-63.888,-179.197,9.160,149.568
C03251=1122.445,184.798,-63.908,-179.195,9.163,149.568
C03252=1122.441,185.013,-63.929,-179.193,9.165,149.569
C03253=1122.436,185.227,-63.949,-179.191,9.167,149.569
C03254=1122.432,185.442,-63.970,-179.188,9.170,149.568
C03255=1122.429,185.654,-63.990,-179.186,9.173,149.568
C03256=1122.425,185.869,-64.011,-179.184,9.175,149.568
C03257=1122.421,186.083,-64.032,-179.182,9.178,149.568
C03258=1122.417,186.332,-64.056,-179.180,9.180,149.569
C03259=1122.412,186.580,-64.080,-179.177,9.183,149.569
C03260=1122.408,186.829,-64.104,-179.175,9.187,149.569
C03261=1122.403,187.078,-64.128,-179.172,9.190,149.569
C03262=1122.398,187.327,-64.152,-179.171,9.192,149.569
C03263=1122.394,187.576,-64.177,-179.168,9.195,149.569
C03264=1122.389,187.824,-64.201,-179.165,9.198,149.569
C03265=1122.385,188.073,-64.225,-179.163,9.200,149.569
C03266=1122.380,188.322,-64.249,-179.161,9.203,149.569
C03267=1122.376,188.570,-64.273,-179.158,9.206,149.569
C03268=1122.371,188.820,-64.298,-179.156,9.209,149.569
C03269=1122.367,189.068,-64.322,-179.154,9.212,149.569
C03270=1122.362,189.317,-64.346,-179.152,9.215,149.569
C03271=1122.357,189.566,-64.370,-179.150,9.218,149.569
C03272=1122.353,189.815,-64.394,-179.148,9.220,149.569
C03273=1122.349,190.063,-64.419,-179.145,9.223,149.569
C03274=1122.344,190.312,-64.443,-179.143,9.225,149.569
C03275=1122.339,190.561,-64.467,-179.141,9.228,149.569
C03276=1122.335,190.810,-64.492,-179.139,9.231,149.569
C03277=1122.330,191.058,-64.516,-179.136,9.234,149.569
C03278=1122.326,191.307,-64.540,-179.135,9.236,149.569
C03279=1122.321,191.556,-64.565,-179.133,9.239,149.570
C03280=1122.317,191.805,-64.590,-179.131,9.242,149.570
C03281=1122.312,192.053,-64.614,-179.129,9.244,149.570
C03282=1122.307,192.302,-64.638,-179.127,9.247,149.570
C03283=1122.304,192.551,-64.663,-179.124,9.250,149.570
C03284=1122.299,192.800,-64.687,-179.123,9.253,149.570
C03285=1122.294,193.048,-64.712,-179.121,9.255,149.570
C03286=1122.290,193.297,-64.737,-179.118,9.258,149.570
C03287=1122.285,193.546,-64.761,-179.117,9.261,149.570
C03288=1122.280,193.795,-64.785,-179.115,9.263,149.570
C03289=1122.276,194.044,-64.810,-179.113,9.265,149.570
C03290=1122.272,194.292,-64.834,-179.111,9.269,149.571
C03291=1122.267,194.541,-64.858,-179.109,9.271,149.571
C03292=1122.263,194.790,-64.883,-179.108,9.274,149.571
C03293=1122.258,195.039,-64.908,-179.106,9.276,149.571
C03294=1122.253,195.287,-64.932,-179.104,9.279,149.571
C03295=1122.249,195.537,-64.957,-179.102,9.281,149.571
C03296=1122.245,195.784,-64.981,-179.101,9.284,149.571
C03297=1122.240,196.034,-65.007,-179.098,9.287,149.572
C03298=1122.236,196.282,-65.031,-179.097,9.290,149.572
C03299=1122.231,196.531,-65.055,-179.094,9.293,149.572
C03300=1122.226,196.780,-65.080,-179.091,9.296,149.572
C03301=1122.222,197.029,-65.104,-179.087,9.300,149.572
C03302=1122.217,197.277,-65.130,-179.084,9.304,149.572
C03303=1122.213,197.526,-65.154,-179.080,9.307,149.571
C03304=1122.208,197.775,-65.179,-179.077,9.311,149.571
C03305=1122.204,198.024,-65.203,-179.073,9.314,149.571
C03306=1122.200,198.237,-65.224,-179.071,9.317,149.571
C03307=1122.197,198.451,-65.246,-179.068,9.320,149.571
C03308=1122.192,198.665,-65.268,-179.065,9.323,149.571
C03309=1122.189,198.879,-65.289,-179.062,9.326,149.571
C03310=1122.184,199.092,-65.311,-179.059,9.329,149.571
C03311=1122.181,199.306,-65.332,-179.056,9.331,149.571
C03312=1122.177,199.520,-65.354,-179.054,9.335,149.571
C03313=1122.173,199.734,-65.375,-179.051,9.337,149.571
C03314=1122.168,199.983,-65.400,-179.047,9.341,149.570
C03315=1122.164,200.231,-65.424,-179.044,9.344,149.570
C03316=1122.160,200.480,-65.449,-179.041,9.347,149.570
C03317=1122.155,200.729,-65.474,-179.038,9.350,149.570
C03318=1122.151,200.977,-65.499,-179.035,9.354,149.570
C03319=1122.146,201.226,-65.524,-179.032,9.356,149.570
C03320=1122.142,201.475,-65.550,-179.029,9.359,149.570
C03321=1122.137,201.724,-65.574,-179.025,9.363,149.570
C03322=1122.133,201.972,-65.600,-179.022,9.365,149.569
C03323=1122.129,202.222,-65.625,-179.019,9.369,149.569
C03324=1122.124,202.470,-65.650,-179.016,9.372,149.569
C03325=1122.119,202.719,-65.675,-179.013,9.375,149.569
C03326=1122.115,202.967,-65.700,-179.010,9.378,149.569
C03327=1122.111,203.216,-65.725,-179.007,9.381,149.569
C03328=1122.106,203.465,-65.750,-179.004,9.384,149.569
C03329=1122.102,203.713,-65.776,-179.001,9.387,149.569
C03330=1122.096,203.962,-65.801,-178.998,9.390,149.569
C03331=1122.093,204.211,-65.826,-178.995,9.392,149.569
C03332=1122.088,204.460,-65.851,-178.992,9.396,149.568
C03333=1122.084,204.708,-65.876,-178.989,9.399,149.568
C03334=1122.079,204.957,-65.902,-178.986,9.402,149.568
C03335=1122.074,205.206,-65.927,-178.983,9.405,149.568
C03336=1122.070,205.454,-65.952,-178.980,9.407,149.568
C03337=1122.066,205.703,-65.978,-178.977,9.410,149.568
C03338=1122.061,205.951,-66.004,-178.975,9.413,149.568
C03339=1122.056,206.201,-66.029,-178.972,9.416,149.568
C03340=1122.052,206.449,-66.053,-178.969,9.419,149.568
C03341=1122.048,206.697,-66.079,-178.966,9.422,149.568
C03342=1122.044,206.946,-66.105,-178.964,9.424,149.568
C03343=1122.039,207.195,-66.130,-178.962,9.427,149.568
C03344=1122.035,207.444,-66.155,-178.959,9.430,149.568
C03345=1122.030,207.692,-66.181,-178.956,9.432,149.567
C03346=1122.026,207.941,-66.206,-178.953,9.435,149.567
C03347=1122.021,208.189,-66.232,-178.950,9.438,149.567
C03348=1122.017,208.438,-66.258,-178.948,9.441,149.567
C03349=1122.012,208.686,-66.283,-178.945,9.443,149.567
C03350=1122.008,208.936,-66.308,-178.943,9.446,149.567
C03351=1122.004,209.185,-66.334,-178.940,9.449,149.567
C03352=1121.999,209.433,-66.359,-178.937,9.452,149.567
C03353=1121.994,209.681,-66.385,-178.935,9.454,149.567
C03354=1121.990,209.930,-66.411,-178.933,9.458,149.567
C03355=1121.985,210.178,-66.436,-178.930,9.460,149.567
C03356=1121.981,210.427,-66.462,-178.928,9.463,149.567
C03357=1121.977,210.676,-66.488,-178.926,9.466,149.567
C03358=1121.973,210.925,-66.514,-178.923,9.469,149.567
C03359=1121.967,211.173,-66.540,-178.921,9.471,149.567
C03360=1121.963,211.422,-66.565,-178.919,9.474,149.567
C03361=1121.959,211.671,-66.591,-178.916,9.477,149.567
C03362=1121.955,211.884,-66.613,-178.914,9.480,149.567
C03363=1121.951,212.098,-66.635,-178.912,9.482,149.568
C03364=1121.948,212.312,-66.658,-178.910,9.484,149.568
C03365=1121.943,212.525,-66.679,-178.909,9.487,149.568
C03366=1121.940,212.739,-66.701,-178.907,9.489,149.568
C03367=1121.935,212.953,-66.724,-178.905,9.491,149.568
C03368=1121.932,213.166,-66.746,-178.903,9.494,149.568
C03369=1121.928,213.380,-66.769,-178.901,9.496,149.568
C03370=1121.924,213.629,-66.794,-178.900,9.499,149.568
C03371=1121.919,213.877,-66.820,-178.897,9.502,149.568
C03372=1121.915,214.126,-66.846,-178.896,9.505,149.568
C03373=1121.910,214.374,-66.871,-178.894,9.507,149.568
C03374=1121.906,214.623,-66.897,-178.892,9.510,149.569
C03375=1121.901,214.872,-66.923,-178.890,9.513,149.569
C03376=1121.897,215.120,-66.950,-178.887,9.516,149.569
C03377=1121.893,215.369,-66.975,-178.886,9.519,149.569
C03378=1121.888,215.617,-67.001,-178.883,9.522,149.569
C03379=1121.884,215.866,-67.027,-178.881,9.524,149.569
C03380=1121.879,216.115,-67.053,-178.879,9.527,149.569
C03381=1121.875,216.364,-67.079,-178.877,9.530,149.569
C03382=1121.871,216.612,-67.105,-178.875,9.533,149.570
C03383=1121.867,216.861,-67.131,-178.873,9.536,149.570
C03384=1121.862,217.109,-67.156,-178.871,9.539,149.570
C03385=1121.857,217.358,-67.183,-178.868,9.542,149.570
C03386=1121.853,217.607,-67.209,-178.866,9.545,149.570
C03387=1121.849,217.855,-67.235,-178.864,9.548,149.570
C03388=1121.844,218.104,-67.262,-178.862,9.551,149.570
C03389=1121.840,218.353,-67.288,-178.859,9.554,149.570
C03390=1121.836,218.601,-67.313,-178.857,9.557,149.570
C03391=1121.831,218.849,-67.340,-178.854,9.560,149.571
C03392=1121.826,219.098,-67.366,-178.852,9.564,149.571
C03393=1121.822,219.347,-67.392,-178.850,9.566,149.571
C03394=1121.818,219.595,-67.418,-178.848,9.569,149.571
C03395=1121.813,219.844,-67.444,-178.845,9.572,149.571
C03396=1121.809,220.092,-67.471,-178.842,9.575,149.571
C03397=1121.805,220.341,-67.497,-178.840,9.579,149.571
C03398=1121.800,220.590,-67.524,-178.838,9.582,149.571
C03399=1121.796,220.838,-67.549,-178.835,9.585,149.571
C03400=1121.792,221.087,-67.575,-178.833,9.588,149.571
C03401=1121.787,221.336,-67.602,-178.830,9.591,149.571
C03402=1121.782,221.584,-67.628,-178.828,9.594,149.572
C03403=1121.778,221.832,-67.655,-178.825,9.597,149.572
C03404=1121.773,222.081,-67.680,-178.823,9.600,149.572
C03405=1121.769,222.330,-67.708,-178.820,9.604,149.572
C03406=1121.765,222.578,-67.734,-178.817,9.607,149.572
C03407=1121.761,222.827,-67.760,-178.814,9.611,149.572
C03408=1121.756,223.075,-67.787,-178.812,9.614,149.572
C03409=1121.752,223.324,-67.813,-178.809,9.616,149.572
C03410=1121.747,223.572,-67.840,-178.806,9.619,149.572
C03411=1121.743,223.821,-67.866,-178.803,9.623,149.572
C03412=1121.738,224.070,-67.892,-178.801,9.626,149.572
C03413=1121.734,224.318,-67.919,-178.798,9.630,149.572
C03414=1121.729,224.567,-67.945,-178.795,9.632,149.572
C03415=1121.725,224.815,-67.972,-178.792,9.636,149.572
C03416=1121.721,225.064,-67.999,-178.790,9.639,149.572
C03417=1121.717,225.312,-68.025,-178.787,9.642,149.572
C03418=1121.713,225.526,-68.048,-178.784,9.645,149.572
C03419=1121.709,225.739,-68.071,-178.782,9.648,149.572
C03420=1121.705,225.953,-68.094,-178.779,9.651,149.572
C03421=1121.701,226.167,-68.117,-178.777,9.653,149.572
C03422=1121.697,226.381,-68.140,-178.774,9.656,149.572
C03423=1121.694,226.594,-68.162,-178.771,9.659,149.572
C03424=1121.690,226.807,-68.185,-178.769,9.662,149.572
C03425=1121.686,227.021,-68.208,-178.766,9.665,149.572
C03426=1121.681,227.269,-68.235,-178.763,9.668,149.572
C03427=1121.678,227.517,-68.262,-178.760,9.672,149.572
C03428=1121.673,227.767,-68.289,-178.757,9.674,149.572
C03429=1121.669,228.016,-68.315,-178.754,9.678,149.572
C03430=1121.665,228.264,-68.342,-178.751,9.681,149.572
C03431=1121.660,228.512,-68.369,-178.747,9.685,149.572
C03432=1121.655,228.761,-68.396,-178.744,9.687,149.571
C03433=1121.651,229.009,-68.422,-178.741,9.691,149.571
C03434=1121.647,229.258,-68.449,-178.738,9.694,149.571
C03435=1121.642,229.506,-68.477,-178.734,9.698,149.571
C03436=1121.638,229.754,-68.503,-178.731,9.701,149.571
C03437=1121.633,230.003,-68.530,-178.728,9.704,149.571
C03438=1121.629,230.252,-68.557,-178.724,9.707,149.571
C03439=1121.625,230.501,-68.585,-178.721,9.711,149.571
C03440=1121.621,230.749,-68.611,-178.718,9.714,149.571
C03441=1121.616,230.997,-68.638,-178.715,9.716,149.571
C03442=1121.612,231.246,-68.665,-178.711,9.720,149.570
C03443=1121.607,231.494,-68.692,-178.708,9.723,149.570
C03444=1121.603,231.743,-68.720,-178.705,9.726,149.570
C03445=1121.599,231.992,-68.746,-178.702,9.729,149.570
C03446=1121.595,232.239,-68.774,-178.699,9.732,149.570
C03447=1121.590,232.488,-68.801,-178.695,9.735,149.570
C03448=1121.585,232.736,-68.828,-178.692,9.738,149.570
C03449=1121.581,232.986,-68.855,-178.689,9.741,149.570
C03450=1121.577,233.234,-68.882,-178.686,9.743,149.569
C03451=1121.573,233.482,-68.909,-178.683,9.746,149.569
C03452=1121.568,233.730,-68.937,-178.680,9.750,149.569
C03453=1121.564,233.979,-68.964,-178.677,9.752,149.569
C03454=1121.560,234.228,-68.991,-178.674,9.755,149.569
C03455=1121.555,234.476,-69.018,-178.671,9.758,149.569
C03456=1121.551,234.724,-69.046,-178.668,9.761,149.569
C03457=1121.546,234.973,-69.073,-178.665,9.763,149.569
C03458=1121.542,235.222,-69.101,-178.662,9.766,149.568
C03459=1121.538,235.470,-69.128,-178.660,9.769,149.569
C03460=1121.534,235.718,-69.155,-178.657,9.772,149.568
C03461=1121.529,235.967,-69.182,-178.654,9.774,149.568
C03462=1121.525,236.215,-69.210,-178.652,9.777,149.568
C03463=1121.520,236.464,-69.237,-178.649,9.779,149.568
C03464=1121.516,236.712,-69.264,-178.646,9.782,149.568
C03465=1121.512,236.961,-69.292,-178.643,9.785,149.568
C03466=1121.507,237.209,-69.319,-178.641,9.787,149.568
C03467=1121.503,237.458,-69.346,-178.638,9.790,149.568
C03468=1121.499,237.706,-69.375,-178.635,9.793,149.568
C03469=1121.494,237.955,-69.402,-178.633,9.795,149.567
C03470=1121.490,238.203,-69.429,-178.630,9.798,149.567
C03471=1121.485,238.451,-69.456,-178.627,9.801,149.567
C03472=1121.482,238.700,-69.485,-178.625,9.803,149.567
C03473=1121.477,238.948,-69.512,-178.622,9.805,149.567
C03474=1121.473,239.162,-69.536,-178.620,9.808,149.567
C03475=1121.469,239.375,-69.560,-178.618,9.810,149.567
C03476=1121.466,239.588,-69.583,-178.616,9.812,149.567
C03477=1121.462,239.802,-69.607,-178.613,9.814,149.567
C03478=1121.458,240.015,-69.631,-178.612,9.816,149.567
C03479=1121.455,240.229,-69.655,-178.609,9.818,149.567
C03480=1121.451,240.443,-69.678,-178.607,9.821,149.567
C03481=1121.446,240.656,-69.702,-178.605,9.823,149.567
C03482=1121.443,240.905,-69.730,-178.603,9.825,149.567
C03483=1121.438,241.152,-69.758,-178.600,9.828,149.567
C03484=1121.434,241.402,-69.785,-178.598,9.830,149.567
C03485=1121.430,241.650,-69.813,-178.596,9.832,149.567
C03486=1121.425,241.898,-69.840,-178.594,9.834,149.567
C03487=1121.421,242.147,-69.868,-178.591,9.837,149.567
C03488=1121.417,242.395,-69.896,-178.589,9.839,149.567
C03489=1121.412,242.643,-69.924,-178.587,9.842,149.567
C03490=1121.408,242.892,-69.952,-178.585,9.844,149.567
C03491=1121.404,243.140,-69.980,-178.582,9.847,149.567
C03492=1121.400,243.389,-70.007,-178.581,9.849,149.567
C03493=1121.395,243.637,-70.035,-178.579,9.851,149.567
C03494=1121.391,243.885,-70.063,-178.577,9.854,149.567
C03495=1121.386,244.134,-70.091,-178.575,9.856,149.567
C03496=1121.382,244.382,-70.118,-178.573,9.858,149.567
C03497=1121.378,244.631,-70.146,-178.571,9.860,149.567
C03498=1121.374,244.879,-70.174,-178.569,9.863,149.567
C03499=1121.369,245.127,-70.203,-178.567,9.865,149.567
C03500=1121.364,245.376,-70.230,-178.565,9.867,149.567
C03501=1121.361,245.625,-70.258,-178.564,9.870,149.567
C03502=1121.356,245.872,-70.286,-178.562,9.872,149.567
C03503=1121.353,246.121,-70.314,-178.560,9.875,149.567
C03504=1121.348,246.369,-70.342,-178.558,9.877,149.567
C03505=1121.343,246.618,-70.370,-178.556,9.879,149.567
C03506=1121.339,246.866,-70.398,-178.554,9.882,149.568
C03507=1121.334,247.114,-70.426,-178.553,9.884,149.568
C03508=1121.330,247.363,-70.454,-178.551,9.887,149.568
C03509=1121.326,247.611,-70.482,-178.547,9.890,149.568
C03510=1121.322,247.859,-70.510,-178.542,9.895,149.567
C03511=1121.317,248.108,-70.538,-178.536,9.899,149.567
C03512=1121.313,248.356,-70.567,-178.531,9.904,149.567
C03513=1121.309,248.605,-70.594,-178.525,9.909,149.566
C03514=1121.304,248.854,-70.622,-178.521,9.912,149.566
C03515=1121.300,249.101,-70.650,-178.516,9.916,149.566
C03516=1121.295,249.350,-70.679,-178.511,9.920,149.565
C03517=1121.292,249.598,-70.708,-178.506,9.924,149.565
C03518=1121.288,249.846,-70.736,-178.502,9.927,149.565
C03519=1121.283,250.095,-70.764,-178.498,9.931,149.564
C03520=1121.279,250.343,-70.792,-178.494,9.934,149.564
C03521=1121.274,250.592,-70.821,-178.490,9.937,149.564
C03522=1121.270,250.840,-70.849,-178.486,9.941,149.564
C03523=1121.265,251.089,-70.877,-178.482,9.943,149.563
C03524=1121.262,251.337,-70.905,-178.478,9.946,149.563
C03525=1121.257,251.585,-70.935,-178.475,9.949,149.563
C03526=1121.253,251.833,-70.963,-178.472,9.951,149.563
C03527=1121.249,252.082,-70.991,-178.469,9.954,149.562
C03528=1121.244,252.330,-71.019,-178.466,9.957,149.562
C03529=1121.240,252.578,-71.049,-178.463,9.958,149.562
C03530=1121.236,252.791,-71.072,-178.462,9.961,149.562
C03531=1121.233,253.005,-71.097,-178.459,9.963,149.562
C03532=1121.229,253.219,-71.122,-178.458,9.964,149.562
C03533=1121.225,253.431,-71.146,-178.456,9.966,149.562
C03534=1121.222,253.645,-71.170,-178.454,9.967,149.562
C03535=1121.218,253.859,-71.196,-178.452,9.970,149.562
C03536=1121.214,254.072,-71.219,-178.450,9.971,149.562
C03537=1121.211,254.285,-71.244,-178.449,9.973,149.562
C03538=1121.206,254.534,-71.273,-178.448,9.974,149.562
C03539=1121.202,254.781,-71.302,-178.447,9.976,149.562
C03540=1121.198,255.030,-71.330,-178.446,9.978,149.562
C03541=1121.194,255.279,-71.358,-178.445,9.979,149.562
C03542=1121.189,255.526,-71.388,-178.444,9.980,149.562
C03543=1121.185,255.775,-71.416,-178.443,9.982,149.562
C03544=1121.181,256.024,-71.444,-178.443,9.983,149.563
C03545=1121.176,256.271,-71.474,-178.440,9.986,149.563
C03546=1121.172,256.520,-71.502,-178.437,9.989,149.562
C03547=1121.168,256.769,-71.530,-178.434,9.992,149.562
C03548=1121.163,257.016,-71.559,-178.432,9.994,149.562
C03549=1121.159,257.265,-71.588,-178.429,9.997,149.562
C03550=1121.155,257.513,-71.617,-178.426,10.000,149.562
C03551=1121.151,257.762,-71.646,-178.423,10.003,149.562
C03552=1121.147,258.009,-71.674,-178.420,10.006,149.562
C03553=1121.142,258.258,-71.703,-178.417,10.009,149.562
C03554=1121.138,258.507,-71.733,-178.414,10.012,149.562
C03555=1121.134,258.754,-71.760,-178.411,10.015,149.562
C03556=1121.130,259.003,-71.790,-178.408,10.018,149.562
C03557=1121.125,259.252,-71.818,-178.405,10.020,149.561
C03558=1121.120,259.572,-71.856,-178.401,10.025,149.561
C03559=1121.114,259.892,-71.893,-178.397,10.028,149.561
C03560=1121.108,260.214,-71.930,-178.393,10.031,149.561
C03561=1121.103,260.535,-71.968,-178.389,10.036,149.561
C03562=1121.099,260.783,-71.997,-178.385,10.038,149.561
C03563=1121.095,261.032,-72.026,-178.383,10.041,149.561
C03564=1121.090,261.279,-72.055,-178.379,10.044,149.560
C03565=1121.086,261.527,-72.084,-178.376,10.047,149.560
C03566=1121.082,261.776,-72.113,-178.373,10.049,149.560
C03567=1121.078,262.024,-72.142,-178.369,10.053,149.560
C03568=1121.074,262.273,-72.172,-178.366,10.056,149.560
C03569=1121.069,262.522,-72.200,-178.363,10.059,149.560
C03570=1121.064,262.769,-72.229,-178.359,10.062,149.560
C03571=1121.060,263.017,-72.259,-178.356,10.064,149.559
C03572=1121.057,263.265,-72.288,-178.352,10.068,149.559
C03573=1121.052,263.514,-72.316,-178.349,10.070,149.559
C03574=1121.048,263.763,-72.346,-178.345,10.074,149.559
C03575=1121.044,264.011,-72.375,-178.342,10.076,149.559
C03576=1121.039,264.258,-72.404,-178.338,10.080,149.558
C03577=1121.035,264.507,-72.434,-178.335,10.082,149.558
C03578=1121.031,264.755,-72.463,-178.333,10.085,149.558
C03579=1121.026,265.004,-72.492,-178.330,10.087,149.558
C03580=1121.022,265.252,-72.522,-178.327,10.090,149.558
C03581=1121.018,265.500,-72.551,-178.325,10.092,149.558
C03582=1121.014,265.749,-72.580,-178.322,10.095,149.558
C03583=1121.009,265.997,-72.610,-178.320,10.096,149.558
C03584=1121.005,266.245,-72.639,-178.317,10.099,149.557
C03585=1121.000,266.493,-72.668,-178.315,10.101,149.557
C03586=1120.995,266.847,-72.710,-178.311,10.105,149.557
C03587=1120.989,267.201,-72.752,-178.306,10.109,149.557
C03588=1120.983,267.554,-72.794,-178.303,10.112,149.557
C03589=1120.977,267.908,-72.836,-178.299,10.115,149.557
C03590=1120.973,268.156,-72.866,-178.296,10.118,149.557
C03591=1120.969,268.405,-72.895,-178.294,10.121,149.557
C03592=1120.964,268.653,-72.925,-178.291,10.123,149.557
C03593=1120.960,268.901,-72.955,-178.288,10.126,149.556
C03594=1120.956,269.150,-72.984,-178.286,10.128,149.556
C03595=1120.951,269.398,-73.014,-178.283,10.131,149.556
C03596=1120.947,269.646,-73.043,-178.280,10.134,149.556
C03597=1120.943,269.894,-73.073,-178.277,10.136,149.556
C03598=1120.939,270.143,-73.102,-178.275,10.138,149.556
C03599=1120.935,270.391,-73.132,-178.272,10.141,149.556
C03600=1120.931,270.639,-73.162,-178.269,10.144,149.556
C03601=1120.927,270.887,-73.191,-178.266,10.147,149.556
C03602=1120.922,271.135,-73.221,-178.262,10.149,149.555
C03603=1120.918,271.384,-73.251,-178.260,10.151,149.555
C03604=1120.913,271.632,-73.280,-178.257,10.154,149.555
C03605=1120.909,271.880,-73.310,-178.254,10.156,149.555
C03606=1120.905,272.128,-73.340,-178.251,10.159,149.555
C03607=1120.901,272.376,-73.369,-178.248,10.162,149.555
C03608=1120.896,272.624,-73.400,-178.245,10.165,149.555
C03609=1120.892,272.872,-73.429,-178.243,10.168,149.555
C03610=1120.888,273.121,-73.459,-178.240,10.170,149.554
C03611=1120.884,273.369,-73.488,-178.237,10.172,149.554
C03612=1120.880,273.617,-73.519,-178.234,10.175,149.554
C03613=1120.875,273.865,-73.549,-178.231,10.177,149.554
C03614=1120.871,274.113,-73.578,-178.228,10.180,149.554
C03615=1120.867,274.361,-73.608,-178.225,10.183,149.554
C03616=1120.863,274.609,-73.638,-178.222,10.186,149.554
C03617=1120.858,274.857,-73.668,-178.219,10.188,149.554
C03618=1120.855,275.106,-73.698,-178.216,10.191,149.553
C03619=1120.851,275.355,-73.728,-178.213,10.194,149.553
C03620=1120.847,275.602,-73.758,-178.210,10.196,149.553
C03621=1120.842,275.851,-73.788,-178.207,10.199,149.553
C03622=1120.838,276.098,-73.818,-178.204,10.202,149.553
C03623=1120.834,276.347,-73.848,-178.201,10.204,149.553
C03624=1120.829,276.595,-73.878,-178.198,10.207,149.552
C03625=1120.825,276.843,-73.908,-178.195,10.210,149.552
C03626=1120.822,277.091,-73.938,-178.192,10.213,149.552
C03627=1120.817,277.340,-73.968,-178.189,10.215,149.552
C03628=1120.813,277.588,-73.999,-178.185,10.219,149.552
C03629=1120.809,277.835,-74.029,-178.182,10.221,149.552
C03630=1120.804,278.084,-74.059,-178.179,10.224,149.552
C03631=1120.800,278.331,-74.089,-178.176,10.227,149.551
C03632=1120.796,278.581,-74.119,-178.173,10.229,149.551
C03633=1120.792,278.828,-74.149,-178.170,10.232,149.551
C03634=1120.788,279.076,-74.180,-178.166,10.234,149.551
C03635=1120.783,279.325,-74.210,-178.163,10.237,149.551
C03636=1120.779,279.572,-74.240,-178.159,10.240,149.550
C03637=1120.775,279.821,-74.271,-178.156,10.243,149.550
C03638=1120.772,280.034,-74.296,-178.154,10.245,149.550
C03639=1120.768,280.247,-74.323,-178.151,10.247,149.550
C03640=1120.764,280.460,-74.349,-178.148,10.250,149.550
C03641=1120.760,280.673,-74.375,-178.146,10.252,149.550
C03642=1120.757,280.886,-74.401,-178.142,10.254,149.549
C03643=1120.754,281.099,-74.427,-178.140,10.256,149.549
C03644=1120.750,281.312,-74.453,-178.137,10.259,149.549
C03645=1120.746,281.525,-74.479,-178.134,10.262,149.549
C03646=1120.742,281.773,-74.509,-178.131,10.264,149.549
C03647=1120.738,282.022,-74.540,-178.128,10.266,149.549
C03648=1120.734,282.270,-74.571,-178.125,10.269,149.548
C03649=1120.729,282.518,-74.601,-178.122,10.271,149.548
C03650=1120.725,282.765,-74.632,-178.119,10.274,149.548
C03651=1120.721,283.015,-74.662,-178.116,10.277,149.548
C03652=1120.717,283.262,-74.692,-178.112,10.279,149.548
C03653=1120.713,283.510,-74.723,-178.110,10.282,149.548
C03654=1120.708,283.758,-74.754,-178.106,10.284,149.547
C03655=1120.705,284.006,-74.784,-178.103,10.287,149.547
C03656=1120.700,284.254,-74.815,-178.101,10.289,149.547
C03657=1120.696,284.502,-74.845,-178.098,10.291,149.547
C03658=1120.692,284.751,-74.876,-178.095,10.294,149.547
C03659=1120.688,284.999,-74.907,-178.091,10.297,149.546
C03660=1120.684,285.246,-74.937,-178.088,10.299,149.546
C03661=1120.680,285.495,-74.968,-178.085,10.302,149.546
C03662=1120.675,285.743,-74.999,-178.082,10.305,149.546
